   Zulauf_RA_V.Tmr_VZ_Anlauf_Q := TRUE;
   Zulauf_RA_V.SS := FALSE;
   Zulauf_RA_V.SSnq := FALSE;
   Zulauf_RA_V.SSfq := TRUE;
   Zulauf_RA_V.nBB := FALSE;
   Zulauf_RA_V.VW_Hand_St1 := FALSE;
   Zulauf_RA_V.VW_Hand_St2 := FALSE;
   Zulauf_RA_V.VW_Hand_Stop := FALSE;
   Zulauf_RA_V.VW_Auto_St1 := FALSE;
   Zulauf_RA_V.VW_Auto_St2 := FALSE;
   Zulauf_RA_V.Anst_Req_St1 := FALSE;
   Zulauf_RA_V.Anst_Req_St2 := FALSE;
   Zulauf_RA_V.FM_Betrieb_Ein := TRUE;
   Zulauf_RA_V.FM_Betrieb_Aus := FALSE;
   Zulauf_RA_V.NLZ_MAZ_St1 := FALSE;
   Zulauf_RA_V.NLZ_MAZ_St2 := FALSE;
   Zulauf_RA_V.NLZ_Rev_SS_St1 := FALSE;
   Zulauf_RA_V.NLZ_Rev_SS_St2 := FALSE;
   Zulauf_RA_V.Th_St := FALSE;
   Zulauf_RA_V.DMA_St := FALSE;
   Zulauf_RA_V.DMZ_St := FALSE;
   Zulauf_RA_V.FU_St := FALSE;
   Zulauf_RA_V.TL_St := FALSE;
   Zulauf_RA_V.UDr_St := FALSE;
   Zulauf_RA_V.UeDr_St := FALSE;
   Zulauf_RA_V.UT_St := FALSE;
   Zulauf_RA_V.Le_St := FALSE;
   Zulauf_RA_V.UeLM_St := FALSE;
   Zulauf_RA_V.UeLE_St := FALSE;
   Zulauf_RA_V.Kom_DP_St := FALSE;
   Zulauf_RA_V.Kom_int_St := FALSE;
   Zulauf_RA_V.int_St := FALSE;
   Zulauf_RA_V.LZ_St := FALSE;
   Zulauf_RA_V.BefLZ_St := FALSE;
   Zulauf_RA_V.FM_GlobalQuit := FALSE;
   Zulauf_RA_V.Quit_RST := FALSE;
   Zulauf_RA_V.Tmr_VZ_Anlauf := 3;
   Zulauf_RA_V.Tmr_VZ_ESZ := 0;
   Zulauf_RA_V.Tmr_Th_St := 0;
   Zulauf_RA_V.Tmr_DMA_St := 0;
   Zulauf_RA_V.Tmr_DMZ_St := 0;
   Zulauf_RA_V.Tmr_FU_St := 0;
   Zulauf_RA_V.Tmr_TL_St := 0;
   Zulauf_RA_V.Tmr_UDr_St := 0;
   Zulauf_RA_V.Tmr_UeDr_St := 0;
   Zulauf_RA_V.Tmr_UT_St := 0;
   Zulauf_RA_V.Tmr_Le_St := 0;
   Zulauf_RA_V.Tmr_UeLM_St := 0;
   Zulauf_RA_V.Tmr_UeLE_St := 0;
   Zulauf_RA_V.Tmr_Kom_DP_St := 0;
   Zulauf_RA_V.Tmr_Kom_int_St := 0;
   Zulauf_RA_V.Tmr_int_St := 0;
   Zulauf_RA_V.Tmr_LZ_St := 0;
   Zulauf_RA_V.Tmr_BefLZ_St := 0;
   Zulauf_RA_V.Tmr_ASZ_St1 := 0;
   Zulauf_RA_V.Tmr_ASZ_St2 := 0;
   Zulauf_RA_V.Tmr_Rev_St1 := 0;
   Zulauf_RA_V.Tmr_Rev_St2 := 0;
   Zulauf_RA_V.BZ_ges_s := 3248;
   Zulauf_RA_V.Tmr_Quit_RST := 0;
   Zulauf_RA_V.BEF_NHV.Bef.Bed_Res := FALSE;
   Zulauf_RA_V.BEF_NHV.Bef.Bed_UV := FALSE;
   Zulauf_RA_V.BEF_NHV.Bef.Bed_NHV := FALSE;
   Zulauf_RA_V.BEF_NHV.Bef.Bed_PLS := FALSE;
   Zulauf_RA_V.BEF_NHV.Bef.BA_Hand := FALSE;
   Zulauf_RA_V.BEF_NHV.Bef.BA_Auto := FALSE;
   Zulauf_RA_V.BEF_NHV.Bef.BF_Ein1 := FALSE;
   Zulauf_RA_V.BEF_NHV.Bef.BF_Ein2 := FALSE;
   Zulauf_RA_V.BEF_NHV.Bef.BF_Aus := FALSE;
   Zulauf_RA_V.BEF_NHV.Bef.BZ_Res := FALSE;
   Zulauf_RA_V.BEF_NHV.Bef.Res_10 := FALSE;
   Zulauf_RA_V.BEF_NHV.Bef.Res_11 := FALSE;
   Zulauf_RA_V.BEF_NHV.Bef.Res_12 := FALSE;
   Zulauf_RA_V.BEF_NHV.Bef.Res_13 := FALSE;
   Zulauf_RA_V.BEF_NHV.Bef.Res_14 := FALSE;
   Zulauf_RA_V.BEF_NHV.Bef.Res_15 := FALSE;
   Zulauf_RA_V.BEF_NHV.Bef.Res_16 := FALSE;
   Zulauf_RA_V.BEF_NHV.Bef.Res_17 := FALSE;
   Zulauf_RA_V.BEF_NHV.Bef.Res_18 := FALSE;
   Zulauf_RA_V.BEF_NHV.Bef.Res_19 := FALSE;
   Zulauf_RA_V.BEF_NHV.Bef.Res_20 := FALSE;
   Zulauf_RA_V.BEF_NHV.Bef.Res_21 := FALSE;
   Zulauf_RA_V.BEF_NHV.Bef.Res_22 := FALSE;
   Zulauf_RA_V.BEF_NHV.Bef.Res_23 := FALSE;
   Zulauf_RA_V.BEF_NHV.Bef.Res_24 := FALSE;
   Zulauf_RA_V.BEF_NHV.Bef.Res_25 := FALSE;
   Zulauf_RA_V.BEF_NHV.Bef.Res_26 := FALSE;
   Zulauf_RA_V.BEF_NHV.Bef.Res_27 := FALSE;
   Zulauf_RA_V.BEF_NHV.Bef.Res_28 := FALSE;
   Zulauf_RA_V.BEF_NHV.Bef.Res_29 := FALSE;
   Zulauf_RA_V.BEF_NHV.Bef.BF_Set_SW_chg := FALSE;
   Zulauf_RA_V.BEF_NHV.Bef.BF_Quit := FALSE;
   Zulauf_RA_V.BEF_NHV.SW_Hand := 0.0;
   Zulauf_RA_RP.Typ := 0;
   Zulauf_RA_RP.Idx := 31;
   Zulauf_RA_RP.BA_VW_Hand := FALSE;
   Zulauf_RA_RP.Tmr_VZ_Anlauf_Q := FALSE;
   Zulauf_RA_RP.SS := FALSE;
   Zulauf_RA_RP.SSnq := FALSE;
   Zulauf_RA_RP.SSfq := TRUE;
   Zulauf_RA_RP.nBB := FALSE;
   Zulauf_RA_RP.VW_Hand_St1 := FALSE;
   Zulauf_RA_RP.VW_Hand_St2 := FALSE;
   Zulauf_RA_RP.VW_Hand_Stop := FALSE;
   Zulauf_RA_RP.VW_Auto_St1 := FALSE;
   Zulauf_RA_RP.VW_Auto_St2 := FALSE;
   Zulauf_RA_RP.Anst_Req_St1 := FALSE;
   Zulauf_RA_RP.Anst_Req_St2 := FALSE;
   Zulauf_RA_RP.FM_Betrieb_Ein := FALSE;
   Zulauf_RA_RP.FM_Betrieb_Aus := TRUE;
   Zulauf_RA_RP.NLZ_MAZ_St1 := FALSE;
   Zulauf_RA_RP.NLZ_MAZ_St2 := FALSE;
   Zulauf_RA_RP.NLZ_Rev_SS_St1 := FALSE;
   Zulauf_RA_RP.NLZ_Rev_SS_St2 := FALSE;
   Zulauf_RA_RP.Th_St := FALSE;
   Zulauf_RA_RP.DMA_St := FALSE;
   Zulauf_RA_RP.DMZ_St := FALSE;
   Zulauf_RA_RP.FU_St := FALSE;
   Zulauf_RA_RP.TL_St := FALSE;
   Zulauf_RA_RP.UDr_St := FALSE;
   Zulauf_RA_RP.UeDr_St := FALSE;
   Zulauf_RA_RP.UT_St := FALSE;
   Zulauf_RA_RP.Le_St := FALSE;
   Zulauf_RA_RP.UeLM_St := FALSE;
   Zulauf_RA_RP.UeLE_St := FALSE;
   Zulauf_RA_RP.Kom_DP_St := FALSE;
   Zulauf_RA_RP.Kom_int_St := FALSE;
   Zulauf_RA_RP.int_St := FALSE;
   Zulauf_RA_RP.LZ_St := FALSE;
   Zulauf_RA_RP.BefLZ_St := FALSE;
   Zulauf_RA_RP.FM_GlobalQuit := FALSE;
   Zulauf_RA_RP.Quit_RST := FALSE;
   Zulauf_RA_RP.Tmr_VZ_Anlauf := 0;
   Zulauf_RA_RP.Tmr_VZ_ESZ := 0;
   Zulauf_RA_RP.Tmr_Th_St := 0;
   Zulauf_RA_RP.Tmr_DMA_St := 0;
   Zulauf_RA_RP.Tmr_DMZ_St := 0;
   Zulauf_RA_RP.Tmr_FU_St := 0;
   Zulauf_RA_RP.Tmr_TL_St := 0;
   Zulauf_RA_RP.Tmr_UDr_St := 0;
   Zulauf_RA_RP.Tmr_UeDr_St := 0;
   Zulauf_RA_RP.Tmr_UT_St := 0;
   Zulauf_RA_RP.Tmr_Le_St := 0;
   Zulauf_RA_RP.Tmr_UeLM_St := 0;
   Zulauf_RA_RP.Tmr_UeLE_St := 0;
   Zulauf_RA_RP.Tmr_Kom_DP_St := 0;
   Zulauf_RA_RP.Tmr_Kom_int_St := 0;
   Zulauf_RA_RP.Tmr_int_St := 0;
   Zulauf_RA_RP.Tmr_LZ_St := 0;
   Zulauf_RA_RP.Tmr_BefLZ_St := 0;
   Zulauf_RA_RP.Tmr_ASZ_St1 := 0;
   Zulauf_RA_RP.Tmr_ASZ_St2 := 0;
   Zulauf_RA_RP.Tmr_Rev_St1 := 0;
   Zulauf_RA_RP.Tmr_Rev_St2 := 0;
   Zulauf_RA_RP.BZ_ges_s := 455;
   Zulauf_RA_RP.Tmr_Quit_RST := 0;
   Zulauf_RA_RP.BEF_NHV.Bef.Bed_Res := FALSE;
   Zulauf_RA_RP.BEF_NHV.Bef.Bed_UV := FALSE;
   Zulauf_RA_RP.BEF_NHV.Bef.Bed_NHV := FALSE;
   Zulauf_RA_RP.BEF_NHV.Bef.Bed_PLS := FALSE;
   Zulauf_RA_RP.BEF_NHV.Bef.BA_Hand := FALSE;
   Zulauf_RA_RP.BEF_NHV.Bef.BA_Auto := FALSE;
   Zulauf_RA_RP.BEF_NHV.Bef.BF_Ein1 := FALSE;
   Zulauf_RA_RP.BEF_NHV.Bef.BF_Ein2 := FALSE;
   Zulauf_RA_RP.BEF_NHV.Bef.BF_Aus := FALSE;
   Zulauf_RA_RP.BEF_NHV.Bef.BZ_Res := FALSE;
   Zulauf_RA_RP.BEF_NHV.Bef.Res_10 := FALSE;
   Zulauf_RA_RP.BEF_NHV.Bef.Res_11 := FALSE;
   Zulauf_RA_RP.BEF_NHV.Bef.Res_12 := FALSE;
   Zulauf_RA_RP.BEF_NHV.Bef.Res_13 := FALSE;
   Zulauf_RA_RP.BEF_NHV.Bef.Res_14 := FALSE;
   Zulauf_RA_RP.BEF_NHV.Bef.Res_15 := FALSE;
   Zulauf_RA_RP.BEF_NHV.Bef.Res_16 := FALSE;
   Zulauf_RA_RP.BEF_NHV.Bef.Res_17 := FALSE;
   Zulauf_RA_RP.BEF_NHV.Bef.Res_18 := FALSE;
   Zulauf_RA_RP.BEF_NHV.Bef.Res_19 := FALSE;
   Zulauf_RA_RP.BEF_NHV.Bef.Res_20 := FALSE;
   Zulauf_RA_RP.BEF_NHV.Bef.Res_21 := FALSE;
   Zulauf_RA_RP.BEF_NHV.Bef.Res_22 := FALSE;
   Zulauf_RA_RP.BEF_NHV.Bef.Res_23 := FALSE;
   Zulauf_RA_RP.BEF_NHV.Bef.Res_24 := FALSE;
   Zulauf_RA_RP.BEF_NHV.Bef.Res_25 := FALSE;
   Zulauf_RA_RP.BEF_NHV.Bef.Res_26 := FALSE;
   Zulauf_RA_RP.BEF_NHV.Bef.Res_27 := FALSE;
   Zulauf_RA_RP.BEF_NHV.Bef.Res_28 := FALSE;
   Zulauf_RA_RP.BEF_NHV.Bef.Res_29 := FALSE;
   Zulauf_RA_RP.BEF_NHV.Bef.BF_Set_SW_chg := FALSE;
   Zulauf_RA_RP.BEF_NHV.Bef.BF_Quit := FALSE;
   Zulauf_RA_RP.BEF_NHV.SW_Hand := 0.0;
   Zulauf_RA_FP.Typ := 0;
   Zulauf_RA_FP.Idx := 32;
   Zulauf_RA_FP.BA_VW_Hand := FALSE;
   Zulauf_RA_FP.Tmr_VZ_Anlauf_Q := FALSE;
   Zulauf_RA_FP.SS := FALSE;
   Zulauf_RA_FP.SSnq := FALSE;
   Zulauf_RA_FP.SSfq := TRUE;
   Zulauf_RA_FP.nBB := FALSE;
   Zulauf_RA_FP.VW_Hand_St1 := FALSE;
   Zulauf_RA_FP.VW_Hand_St2 := FALSE;
   Zulauf_RA_FP.VW_Hand_Stop := FALSE;
   Zulauf_RA_FP.VW_Auto_St1 := FALSE;
   Zulauf_RA_FP.VW_Auto_St2 := FALSE;
   Zulauf_RA_FP.Anst_Req_St1 := FALSE;
   Zulauf_RA_FP.Anst_Req_St2 := FALSE;
   Zulauf_RA_FP.FM_Betrieb_Ein := FALSE;
   Zulauf_RA_FP.FM_Betrieb_Aus := TRUE;
   Zulauf_RA_FP.NLZ_MAZ_St1 := FALSE;
   Zulauf_RA_FP.NLZ_MAZ_St2 := FALSE;
   Zulauf_RA_FP.NLZ_Rev_SS_St1 := FALSE;
   Zulauf_RA_FP.NLZ_Rev_SS_St2 := FALSE;
   Zulauf_RA_FP.Th_St := FALSE;
   Zulauf_RA_FP.DMA_St := FALSE;
   Zulauf_RA_FP.DMZ_St := FALSE;
   Zulauf_RA_FP.FU_St := FALSE;
   Zulauf_RA_FP.TL_St := FALSE;
   Zulauf_RA_FP.UDr_St := FALSE;
   Zulauf_RA_FP.UeDr_St := FALSE;
   Zulauf_RA_FP.UT_St := FALSE;
   Zulauf_RA_FP.Le_St := FALSE;
   Zulauf_RA_FP.UeLM_St := FALSE;
   Zulauf_RA_FP.UeLE_St := FALSE;
   Zulauf_RA_FP.Kom_DP_St := FALSE;
   Zulauf_RA_FP.Kom_int_St := FALSE;
   Zulauf_RA_FP.int_St := FALSE;
   Zulauf_RA_FP.LZ_St := FALSE;
   Zulauf_RA_FP.BefLZ_St := FALSE;
   Zulauf_RA_FP.FM_GlobalQuit := FALSE;
   Zulauf_RA_FP.Quit_RST := FALSE;
   Zulauf_RA_FP.Tmr_VZ_Anlauf := 0;
   Zulauf_RA_FP.Tmr_VZ_ESZ := 0;
   Zulauf_RA_FP.Tmr_Th_St := 0;
   Zulauf_RA_FP.Tmr_DMA_St := 0;
   Zulauf_RA_FP.Tmr_DMZ_St := 0;
   Zulauf_RA_FP.Tmr_FU_St := 0;
   Zulauf_RA_FP.Tmr_TL_St := 0;
   Zulauf_RA_FP.Tmr_UDr_St := 0;
   Zulauf_RA_FP.Tmr_UeDr_St := 0;
   Zulauf_RA_FP.Tmr_UT_St := 0;
   Zulauf_RA_FP.Tmr_Le_St := 0;
   Zulauf_RA_FP.Tmr_UeLM_St := 0;
   Zulauf_RA_FP.Tmr_UeLE_St := 0;
   Zulauf_RA_FP.Tmr_Kom_DP_St := 0;
   Zulauf_RA_FP.Tmr_Kom_int_St := 0;
   Zulauf_RA_FP.Tmr_int_St := 0;
   Zulauf_RA_FP.Tmr_LZ_St := 0;
   Zulauf_RA_FP.Tmr_BefLZ_St := 0;
   Zulauf_RA_FP.Tmr_ASZ_St1 := 0;
   Zulauf_RA_FP.Tmr_ASZ_St2 := 0;
   Zulauf_RA_FP.Tmr_Rev_St1 := 0;
   Zulauf_RA_FP.Tmr_Rev_St2 := 0;
   Zulauf_RA_FP.BZ_ges_s := 701;
   Zulauf_RA_FP.Tmr_Quit_RST := 0;
   Zulauf_RA_FP.BEF_NHV.Bef.Bed_Res := FALSE;
   Zulauf_RA_FP.BEF_NHV.Bef.Bed_UV := FALSE;
   Zulauf_RA_FP.BEF_NHV.Bef.Bed_NHV := FALSE;
   Zulauf_RA_FP.BEF_NHV.Bef.Bed_PLS := FALSE;
   Zulauf_RA_FP.BEF_NHV.Bef.BA_Hand := FALSE;
   Zulauf_RA_FP.BEF_NHV.Bef.BA_Auto := FALSE;
   Zulauf_RA_FP.BEF_NHV.Bef.BF_Ein1 := FALSE;
   Zulauf_RA_FP.BEF_NHV.Bef.BF_Ein2 := FALSE;
   Zulauf_RA_FP.BEF_NHV.Bef.BF_Aus := FALSE;
   Zulauf_RA_FP.BEF_NHV.Bef.BZ_Res := FALSE;
   Zulauf_RA_FP.BEF_NHV.Bef.Res_10 := FALSE;
   Zulauf_RA_FP.BEF_NHV.Bef.Res_11 := FALSE;
   Zulauf_RA_FP.BEF_NHV.Bef.Res_12 := FALSE;
   Zulauf_RA_FP.BEF_NHV.Bef.Res_13 := FALSE;
   Zulauf_RA_FP.BEF_NHV.Bef.Res_14 := FALSE;
   Zulauf_RA_FP.BEF_NHV.Bef.Res_15 := FALSE;
   Zulauf_RA_FP.BEF_NHV.Bef.Res_16 := FALSE;
   Zulauf_RA_FP.BEF_NHV.Bef.Res_17 := FALSE;
   Zulauf_RA_FP.BEF_NHV.Bef.Res_18 := FALSE;
   Zulauf_RA_FP.BEF_NHV.Bef.Res_19 := FALSE;
   Zulauf_RA_FP.BEF_NHV.Bef.Res_20 := FALSE;
   Zulauf_RA_FP.BEF_NHV.Bef.Res_21 := FALSE;
   Zulauf_RA_FP.BEF_NHV.Bef.Res_22 := FALSE;
   Zulauf_RA_FP.BEF_NHV.Bef.Res_23 := FALSE;
   Zulauf_RA_FP.BEF_NHV.Bef.Res_24 := FALSE;
   Zulauf_RA_FP.BEF_NHV.Bef.Res_25 := FALSE;
   Zulauf_RA_FP.BEF_NHV.Bef.Res_26 := FALSE;
   Zulauf_RA_FP.BEF_NHV.Bef.Res_27 := FALSE;
   Zulauf_RA_FP.BEF_NHV.Bef.Res_28 := FALSE;
   Zulauf_RA_FP.BEF_NHV.Bef.Res_29 := FALSE;
   Zulauf_RA_FP.BEF_NHV.Bef.BF_Set_SW_chg := FALSE;
   Zulauf_RA_FP.BEF_NHV.Bef.BF_Quit := FALSE;
   Zulauf_RA_FP.BEF_NHV.SW_Hand := 0.0;
   Schlamm_BP.Typ := 0;
   Schlamm_BP.Idx := 33;
   Schlamm_BP.BA_VW_Hand := FALSE;
   Schlamm_BP.Tmr_VZ_Anlauf_Q := FALSE;
   Schlamm_BP.SS := FALSE;
   Schlamm_BP.SSnq := FALSE;
   Schlamm_BP.SSfq := TRUE;
   Schlamm_BP.nBB := FALSE;
   Schlamm_BP.VW_Hand_St1 := FALSE;
   Schlamm_BP.VW_Hand_St2 := FALSE;
   Schlamm_BP.VW_Hand_Stop := FALSE;
   Schlamm_BP.VW_Auto_St1 := FALSE;
   Schlamm_BP.VW_Auto_St2 := FALSE;
   Schlamm_BP.Anst_Req_St1 := FALSE;
   Schlamm_BP.Anst_Req_St2 := FALSE;
   Schlamm_BP.FM_Betrieb_Ein := FALSE;
   Schlamm_BP.FM_Betrieb_Aus := TRUE;
   Schlamm_BP.NLZ_MAZ_St1 := FALSE;
   Schlamm_BP.NLZ_MAZ_St2 := FALSE;
   Schlamm_BP.NLZ_Rev_SS_St1 := FALSE;
   Schlamm_BP.NLZ_Rev_SS_St2 := FALSE;
   Schlamm_BP.Th_St := FALSE;
   Schlamm_BP.DMA_St := FALSE;
   Schlamm_BP.DMZ_St := FALSE;
   Schlamm_BP.FU_St := FALSE;
   Schlamm_BP.TL_St := FALSE;
   Schlamm_BP.UDr_St := FALSE;
   Schlamm_BP.UeDr_St := FALSE;
   Schlamm_BP.UT_St := FALSE;
   Schlamm_BP.Le_St := FALSE;
   Schlamm_BP.UeLM_St := FALSE;
   Schlamm_BP.UeLE_St := FALSE;
   Schlamm_BP.Kom_DP_St := FALSE;
   Schlamm_BP.Kom_int_St := FALSE;
   Schlamm_BP.int_St := FALSE;
   Schlamm_BP.LZ_St := FALSE;
   Schlamm_BP.BefLZ_St := FALSE;
   Schlamm_BP.FM_GlobalQuit := FALSE;
   Schlamm_BP.Quit_RST := FALSE;
   Schlamm_BP.Tmr_VZ_Anlauf := 0;
   Schlamm_BP.Tmr_VZ_ESZ := 0;
   Schlamm_BP.Tmr_Th_St := 0;
   Schlamm_BP.Tmr_DMA_St := 0;
   Schlamm_BP.Tmr_DMZ_St := 0;
   Schlamm_BP.Tmr_FU_St := 0;
   Schlamm_BP.Tmr_TL_St := 0;
   Schlamm_BP.Tmr_UDr_St := 0;
   Schlamm_BP.Tmr_UeDr_St := 0;
   Schlamm_BP.Tmr_UT_St := 0;
   Schlamm_BP.Tmr_Le_St := 0;
   Schlamm_BP.Tmr_UeLM_St := 0;
   Schlamm_BP.Tmr_UeLE_St := 0;
   Schlamm_BP.Tmr_Kom_DP_St := 0;
   Schlamm_BP.Tmr_Kom_int_St := 0;
   Schlamm_BP.Tmr_int_St := 0;
   Schlamm_BP.Tmr_LZ_St := 0;
   Schlamm_BP.Tmr_BefLZ_St := 0;
   Schlamm_BP.Tmr_ASZ_St1 := 0;
   Schlamm_BP.Tmr_ASZ_St2 := 0;
   Schlamm_BP.Tmr_Rev_St1 := 0;
   Schlamm_BP.Tmr_Rev_St2 := 0;
   Schlamm_BP.BZ_ges_s := 708;
   Schlamm_BP.Tmr_Quit_RST := 0;
   Schlamm_BP.BEF_NHV.Bef.Bed_Res := FALSE;
   Schlamm_BP.BEF_NHV.Bef.Bed_UV := FALSE;
   Schlamm_BP.BEF_NHV.Bef.Bed_NHV := FALSE;
   Schlamm_BP.BEF_NHV.Bef.Bed_PLS := FALSE;
   Schlamm_BP.BEF_NHV.Bef.BA_Hand := FALSE;
   Schlamm_BP.BEF_NHV.Bef.BA_Auto := FALSE;
   Schlamm_BP.BEF_NHV.Bef.BF_Ein1 := FALSE;
   Schlamm_BP.BEF_NHV.Bef.BF_Ein2 := FALSE;
   Schlamm_BP.BEF_NHV.Bef.BF_Aus := FALSE;
   Schlamm_BP.BEF_NHV.Bef.BZ_Res := FALSE;
   Schlamm_BP.BEF_NHV.Bef.Res_10 := FALSE;
   Schlamm_BP.BEF_NHV.Bef.Res_11 := FALSE;
   Schlamm_BP.BEF_NHV.Bef.Res_12 := FALSE;
   Schlamm_BP.BEF_NHV.Bef.Res_13 := FALSE;
   Schlamm_BP.BEF_NHV.Bef.Res_14 := FALSE;
   Schlamm_BP.BEF_NHV.Bef.Res_15 := FALSE;
   Schlamm_BP.BEF_NHV.Bef.Res_16 := FALSE;
   Schlamm_BP.BEF_NHV.Bef.Res_17 := FALSE;
   Schlamm_BP.BEF_NHV.Bef.Res_18 := FALSE;
   Schlamm_BP.BEF_NHV.Bef.Res_19 := FALSE;
   Schlamm_BP.BEF_NHV.Bef.Res_20 := FALSE;
   Schlamm_BP.BEF_NHV.Bef.Res_21 := FALSE;
   Schlamm_BP.BEF_NHV.Bef.Res_22 := FALSE;
   Schlamm_BP.BEF_NHV.Bef.Res_23 := FALSE;
   Schlamm_BP.BEF_NHV.Bef.Res_24 := FALSE;
   Schlamm_BP.BEF_NHV.Bef.Res_25 := FALSE;
   Schlamm_BP.BEF_NHV.Bef.Res_26 := FALSE;
   Schlamm_BP.BEF_NHV.Bef.Res_27 := FALSE;
   Schlamm_BP.BEF_NHV.Bef.Res_28 := FALSE;
   Schlamm_BP.BEF_NHV.Bef.Res_29 := FALSE;
   Schlamm_BP.BEF_NHV.Bef.BF_Set_SW_chg := FALSE;
   Schlamm_BP.BEF_NHV.Bef.BF_Quit := FALSE;
   Schlamm_BP.BEF_NHV.SW_Hand := 0.0;
   Truebwasser_P1.Typ := 0;
   Truebwasser_P1.Idx := 34;
   Truebwasser_P1.BA_VW_Hand := FALSE;
   Truebwasser_P1.Tmr_VZ_Anlauf_Q := FALSE;
   Truebwasser_P1.SS := FALSE;
   Truebwasser_P1.SSnq := FALSE;
   Truebwasser_P1.SSfq := TRUE;
   Truebwasser_P1.nBB := FALSE;
   Truebwasser_P1.VW_Hand_St1 := FALSE;
   Truebwasser_P1.VW_Hand_St2 := FALSE;
   Truebwasser_P1.VW_Hand_Stop := FALSE;
   Truebwasser_P1.VW_Auto_St1 := FALSE;
   Truebwasser_P1.VW_Auto_St2 := FALSE;
   Truebwasser_P1.Anst_Req_St1 := FALSE;
   Truebwasser_P1.Anst_Req_St2 := FALSE;
   Truebwasser_P1.FM_Betrieb_Ein := FALSE;
   Truebwasser_P1.FM_Betrieb_Aus := TRUE;
   Truebwasser_P1.NLZ_MAZ_St1 := FALSE;
   Truebwasser_P1.NLZ_MAZ_St2 := FALSE;
   Truebwasser_P1.NLZ_Rev_SS_St1 := FALSE;
   Truebwasser_P1.NLZ_Rev_SS_St2 := FALSE;
   Truebwasser_P1.Th_St := FALSE;
   Truebwasser_P1.DMA_St := FALSE;
   Truebwasser_P1.DMZ_St := FALSE;
   Truebwasser_P1.FU_St := FALSE;
   Truebwasser_P1.TL_St := FALSE;
   Truebwasser_P1.UDr_St := FALSE;
   Truebwasser_P1.UeDr_St := FALSE;
   Truebwasser_P1.UT_St := FALSE;
   Truebwasser_P1.Le_St := FALSE;
   Truebwasser_P1.UeLM_St := FALSE;
   Truebwasser_P1.UeLE_St := FALSE;
   Truebwasser_P1.Kom_DP_St := FALSE;
   Truebwasser_P1.Kom_int_St := FALSE;
   Truebwasser_P1.int_St := FALSE;
   Truebwasser_P1.LZ_St := FALSE;
   Truebwasser_P1.BefLZ_St := FALSE;
   Truebwasser_P1.FM_GlobalQuit := FALSE;
   Truebwasser_P1.Quit_RST := FALSE;
   Truebwasser_P1.Tmr_VZ_Anlauf := 0;
   Truebwasser_P1.Tmr_VZ_ESZ := 0;
   Truebwasser_P1.Tmr_Th_St := 0;
   Truebwasser_P1.Tmr_DMA_St := 0;
   Truebwasser_P1.Tmr_DMZ_St := 0;
   Truebwasser_P1.Tmr_FU_St := 0;
   Truebwasser_P1.Tmr_TL_St := 0;
   Truebwasser_P1.Tmr_UDr_St := 0;
   Truebwasser_P1.Tmr_UeDr_St := 0;
   Truebwasser_P1.Tmr_UT_St := 0;
   Truebwasser_P1.Tmr_Le_St := 0;
   Truebwasser_P1.Tmr_UeLM_St := 0;
   Truebwasser_P1.Tmr_UeLE_St := 0;
   Truebwasser_P1.Tmr_Kom_DP_St := 0;
   Truebwasser_P1.Tmr_Kom_int_St := 0;
   Truebwasser_P1.Tmr_int_St := 0;
   Truebwasser_P1.Tmr_LZ_St := 0;
   Truebwasser_P1.Tmr_BefLZ_St := 0;
   Truebwasser_P1.Tmr_ASZ_St1 := 0;
   Truebwasser_P1.Tmr_ASZ_St2 := 0;
   Truebwasser_P1.Tmr_Rev_St1 := 0;
   Truebwasser_P1.Tmr_Rev_St2 := 0;
   Truebwasser_P1.BZ_ges_s := 842;
   Truebwasser_P1.Tmr_Quit_RST := 0;
   Truebwasser_P1.BEF_NHV.Bef.Bed_Res := FALSE;
   Truebwasser_P1.BEF_NHV.Bef.Bed_UV := FALSE;
   Truebwasser_P1.BEF_NHV.Bef.Bed_NHV := FALSE;
   Truebwasser_P1.BEF_NHV.Bef.Bed_PLS := FALSE;
   Truebwasser_P1.BEF_NHV.Bef.BA_Hand := FALSE;
   Truebwasser_P1.BEF_NHV.Bef.BA_Auto := FALSE;
   Truebwasser_P1.BEF_NHV.Bef.BF_Ein1 := FALSE;
   Truebwasser_P1.BEF_NHV.Bef.BF_Ein2 := FALSE;
   Truebwasser_P1.BEF_NHV.Bef.BF_Aus := FALSE;
   Truebwasser_P1.BEF_NHV.Bef.BZ_Res := FALSE;
   Truebwasser_P1.BEF_NHV.Bef.Res_10 := FALSE;
   Truebwasser_P1.BEF_NHV.Bef.Res_11 := FALSE;
   Truebwasser_P1.BEF_NHV.Bef.Res_12 := FALSE;
   Truebwasser_P1.BEF_NHV.Bef.Res_13 := FALSE;
   Truebwasser_P1.BEF_NHV.Bef.Res_14 := FALSE;
   Truebwasser_P1.BEF_NHV.Bef.Res_15 := FALSE;
   Truebwasser_P1.BEF_NHV.Bef.Res_16 := FALSE;
   Truebwasser_P1.BEF_NHV.Bef.Res_17 := FALSE;
   Truebwasser_P1.BEF_NHV.Bef.Res_18 := FALSE;
   Truebwasser_P1.BEF_NHV.Bef.Res_19 := FALSE;
   Truebwasser_P1.BEF_NHV.Bef.Res_20 := FALSE;
   Truebwasser_P1.BEF_NHV.Bef.Res_21 := FALSE;
   Truebwasser_P1.BEF_NHV.Bef.Res_22 := FALSE;
   Truebwasser_P1.BEF_NHV.Bef.Res_23 := FALSE;
   Truebwasser_P1.BEF_NHV.Bef.Res_24 := FALSE;
   Truebwasser_P1.BEF_NHV.Bef.Res_25 := FALSE;
   Truebwasser_P1.BEF_NHV.Bef.Res_26 := FALSE;
   Truebwasser_P1.BEF_NHV.Bef.Res_27 := FALSE;
   Truebwasser_P1.BEF_NHV.Bef.Res_28 := FALSE;
   Truebwasser_P1.BEF_NHV.Bef.Res_29 := FALSE;
   Truebwasser_P1.BEF_NHV.Bef.BF_Set_SW_chg := FALSE;
   Truebwasser_P1.BEF_NHV.Bef.BF_Quit := FALSE;
   Truebwasser_P1.BEF_NHV.SW_Hand := 0.0;
   Truebwasser_P2.Typ := 0;
   Truebwasser_P2.Idx := 35;
   Truebwasser_P2.BA_VW_Hand := FALSE;
   Truebwasser_P2.Tmr_VZ_Anlauf_Q := FALSE;
   Truebwasser_P2.SS := FALSE;
   Truebwasser_P2.SSnq := FALSE;
   Truebwasser_P2.SSfq := TRUE;
   Truebwasser_P2.nBB := FALSE;
   Truebwasser_P2.VW_Hand_St1 := FALSE;
   Truebwasser_P2.VW_Hand_St2 := FALSE;
   Truebwasser_P2.VW_Hand_Stop := FALSE;
   Truebwasser_P2.VW_Auto_St1 := FALSE;
   Truebwasser_P2.VW_Auto_St2 := FALSE;
   Truebwasser_P2.Anst_Req_St1 := FALSE;
   Truebwasser_P2.Anst_Req_St2 := FALSE;
   Truebwasser_P2.FM_Betrieb_Ein := FALSE;
   Truebwasser_P2.FM_Betrieb_Aus := TRUE;
   Truebwasser_P2.NLZ_MAZ_St1 := FALSE;
   Truebwasser_P2.NLZ_MAZ_St2 := FALSE;
   Truebwasser_P2.NLZ_Rev_SS_St1 := FALSE;
   Truebwasser_P2.NLZ_Rev_SS_St2 := FALSE;
   Truebwasser_P2.Th_St := FALSE;
   Truebwasser_P2.DMA_St := FALSE;
   Truebwasser_P2.DMZ_St := FALSE;
   Truebwasser_P2.FU_St := FALSE;
   Truebwasser_P2.TL_St := FALSE;
   Truebwasser_P2.UDr_St := FALSE;
   Truebwasser_P2.UeDr_St := FALSE;
   Truebwasser_P2.UT_St := FALSE;
   Truebwasser_P2.Le_St := FALSE;
   Truebwasser_P2.UeLM_St := FALSE;
   Truebwasser_P2.UeLE_St := FALSE;
   Truebwasser_P2.Kom_DP_St := FALSE;
   Truebwasser_P2.Kom_int_St := FALSE;
   Truebwasser_P2.int_St := FALSE;
   Truebwasser_P2.LZ_St := FALSE;
   Truebwasser_P2.BefLZ_St := FALSE;
   Truebwasser_P2.FM_GlobalQuit := FALSE;
   Truebwasser_P2.Quit_RST := FALSE;
   Truebwasser_P2.Tmr_VZ_Anlauf := 0;
   Truebwasser_P2.Tmr_VZ_ESZ := 0;
   Truebwasser_P2.Tmr_Th_St := 0;
   Truebwasser_P2.Tmr_DMA_St := 0;
   Truebwasser_P2.Tmr_DMZ_St := 0;
   Truebwasser_P2.Tmr_FU_St := 0;
   Truebwasser_P2.Tmr_TL_St := 0;
   Truebwasser_P2.Tmr_UDr_St := 0;
   Truebwasser_P2.Tmr_UeDr_St := 0;
   Truebwasser_P2.Tmr_UT_St := 0;
   Truebwasser_P2.Tmr_Le_St := 0;
   Truebwasser_P2.Tmr_UeLM_St := 0;
   Truebwasser_P2.Tmr_UeLE_St := 0;
   Truebwasser_P2.Tmr_Kom_DP_St := 0;
   Truebwasser_P2.Tmr_Kom_int_St := 0;
   Truebwasser_P2.Tmr_int_St := 0;
   Truebwasser_P2.Tmr_LZ_St := 0;
   Truebwasser_P2.Tmr_BefLZ_St := 0;
   Truebwasser_P2.Tmr_ASZ_St1 := 0;
   Truebwasser_P2.Tmr_ASZ_St2 := 0;
   Truebwasser_P2.Tmr_Rev_St1 := 0;
   Truebwasser_P2.Tmr_Rev_St2 := 0;
   Truebwasser_P2.BZ_ges_s := 1903;
   Truebwasser_P2.Tmr_Quit_RST := 0;
   Truebwasser_P2.BEF_NHV.Bef.Bed_Res := FALSE;
   Truebwasser_P2.BEF_NHV.Bef.Bed_UV := FALSE;
   Truebwasser_P2.BEF_NHV.Bef.Bed_NHV := FALSE;
   Truebwasser_P2.BEF_NHV.Bef.Bed_PLS := FALSE;
   Truebwasser_P2.BEF_NHV.Bef.BA_Hand := FALSE;
   Truebwasser_P2.BEF_NHV.Bef.BA_Auto := FALSE;
   Truebwasser_P2.BEF_NHV.Bef.BF_Ein1 := FALSE;
   Truebwasser_P2.BEF_NHV.Bef.BF_Ein2 := FALSE;
   Truebwasser_P2.BEF_NHV.Bef.BF_Aus := FALSE;
   Truebwasser_P2.BEF_NHV.Bef.BZ_Res := FALSE;
   Truebwasser_P2.BEF_NHV.Bef.Res_10 := FALSE;
   Truebwasser_P2.BEF_NHV.Bef.Res_11 := FALSE;
   Truebwasser_P2.BEF_NHV.Bef.Res_12 := FALSE;
   Truebwasser_P2.BEF_NHV.Bef.Res_13 := FALSE;
   Truebwasser_P2.BEF_NHV.Bef.Res_14 := FALSE;
   Truebwasser_P2.BEF_NHV.Bef.Res_15 := FALSE;
   Truebwasser_P2.BEF_NHV.Bef.Res_16 := FALSE;
   Truebwasser_P2.BEF_NHV.Bef.Res_17 := FALSE;
   Truebwasser_P2.BEF_NHV.Bef.Res_18 := FALSE;
   Truebwasser_P2.BEF_NHV.Bef.Res_19 := FALSE;
   Truebwasser_P2.BEF_NHV.Bef.Res_20 := FALSE;
   Truebwasser_P2.BEF_NHV.Bef.Res_21 := FALSE;
   Truebwasser_P2.BEF_NHV.Bef.Res_22 := FALSE;
   Truebwasser_P2.BEF_NHV.Bef.Res_23 := FALSE;
   Truebwasser_P2.BEF_NHV.Bef.Res_24 := FALSE;
   Truebwasser_P2.BEF_NHV.Bef.Res_25 := FALSE;
   Truebwasser_P2.BEF_NHV.Bef.Res_26 := FALSE;
   Truebwasser_P2.BEF_NHV.Bef.Res_27 := FALSE;
   Truebwasser_P2.BEF_NHV.Bef.Res_28 := FALSE;
   Truebwasser_P2.BEF_NHV.Bef.Res_29 := FALSE;
   Truebwasser_P2.BEF_NHV.Bef.BF_Set_SW_chg := FALSE;
   Truebwasser_P2.BEF_NHV.Bef.BF_Quit := FALSE;
   Truebwasser_P2.BEF_NHV.SW_Hand := 0.0;
   Schlamm_AS.Typ := 5;
   Schlamm_AS.Idx := 36;
   Schlamm_AS.BA_VW_Hand := FALSE;
   Schlamm_AS.Tmr_VZ_Anlauf_Q := FALSE;
   Schlamm_AS.SS := FALSE;
   Schlamm_AS.SSnq := FALSE;
   Schlamm_AS.SSfq := TRUE;
   Schlamm_AS.nBB := FALSE;
   Schlamm_AS.VW_Hand_St1 := FALSE;
   Schlamm_AS.VW_Hand_St2 := FALSE;
   Schlamm_AS.VW_Hand_Stop := FALSE;
   Schlamm_AS.VW_Auto_St1 := FALSE;
   Schlamm_AS.VW_Auto_St2 := FALSE;
   Schlamm_AS.Anst_Req_St1 := FALSE;
   Schlamm_AS.Anst_Req_St2 := FALSE;
   Schlamm_AS.FM_Betrieb_Ein := FALSE;
   Schlamm_AS.FM_Betrieb_Aus := TRUE;
   Schlamm_AS.NLZ_MAZ_St1 := FALSE;
   Schlamm_AS.NLZ_MAZ_St2 := FALSE;
   Schlamm_AS.NLZ_Rev_SS_St1 := FALSE;
   Schlamm_AS.NLZ_Rev_SS_St2 := FALSE;
   Schlamm_AS.Th_St := FALSE;
   Schlamm_AS.DMA_St := FALSE;
   Schlamm_AS.DMZ_St := FALSE;
   Schlamm_AS.FU_St := FALSE;
   Schlamm_AS.TL_St := FALSE;
   Schlamm_AS.UDr_St := FALSE;
   Schlamm_AS.UeDr_St := FALSE;
   Schlamm_AS.UT_St := FALSE;
   Schlamm_AS.Le_St := FALSE;
   Schlamm_AS.UeLM_St := FALSE;
   Schlamm_AS.UeLE_St := FALSE;
   Schlamm_AS.Kom_DP_St := FALSE;
   Schlamm_AS.Kom_int_St := FALSE;
   Schlamm_AS.int_St := FALSE;
   Schlamm_AS.LZ_St := FALSE;
   Schlamm_AS.BefLZ_St := FALSE;
   Schlamm_AS.FM_GlobalQuit := FALSE;
   Schlamm_AS.Quit_RST := FALSE;
   Schlamm_AS.Tmr_VZ_Anlauf := 0;
   Schlamm_AS.Tmr_VZ_ESZ := 0;
   Schlamm_AS.Tmr_Th_St := 0;
   Schlamm_AS.Tmr_DMA_St := 0;
   Schlamm_AS.Tmr_DMZ_St := 0;
   Schlamm_AS.Tmr_FU_St := 0;
   Schlamm_AS.Tmr_TL_St := 0;
   Schlamm_AS.Tmr_UDr_St := 0;
   Schlamm_AS.Tmr_UeDr_St := 0;
   Schlamm_AS.Tmr_UT_St := 0;
   Schlamm_AS.Tmr_Le_St := 0;
   Schlamm_AS.Tmr_UeLM_St := 0;
   Schlamm_AS.Tmr_UeLE_St := 0;
   Schlamm_AS.Tmr_Kom_DP_St := 0;
   Schlamm_AS.Tmr_Kom_int_St := 0;
   Schlamm_AS.Tmr_int_St := 0;
   Schlamm_AS.Tmr_LZ_St := 0;
   Schlamm_AS.Tmr_BefLZ_St := 0;
   Schlamm_AS.Tmr_ASZ_St1 := 0;
   Schlamm_AS.Tmr_ASZ_St2 := 0;
   Schlamm_AS.Tmr_Rev_St1 := 0;
   Schlamm_AS.Tmr_Rev_St2 := 0;
   Schlamm_AS.BZ_ges_s := 139;
   Schlamm_AS.Tmr_Quit_RST := 0;
   Schlamm_AS.BEF_NHV.Bef.Bed_Res := FALSE;
   Schlamm_AS.BEF_NHV.Bef.Bed_UV := FALSE;
   Schlamm_AS.BEF_NHV.Bef.Bed_NHV := FALSE;
   Schlamm_AS.BEF_NHV.Bef.Bed_PLS := FALSE;
   Schlamm_AS.BEF_NHV.Bef.BA_Hand := FALSE;
   Schlamm_AS.BEF_NHV.Bef.BA_Auto := FALSE;
   Schlamm_AS.BEF_NHV.Bef.BF_Ein1 := FALSE;
   Schlamm_AS.BEF_NHV.Bef.BF_Ein2 := FALSE;
   Schlamm_AS.BEF_NHV.Bef.BF_Aus := FALSE;
   Schlamm_AS.BEF_NHV.Bef.BZ_Res := FALSE;
   Schlamm_AS.BEF_NHV.Bef.Res_10 := FALSE;
   Schlamm_AS.BEF_NHV.Bef.Res_11 := FALSE;
   Schlamm_AS.BEF_NHV.Bef.Res_12 := FALSE;
   Schlamm_AS.BEF_NHV.Bef.Res_13 := FALSE;
   Schlamm_AS.BEF_NHV.Bef.Res_14 := FALSE;
   Schlamm_AS.BEF_NHV.Bef.Res_15 := FALSE;
   Schlamm_AS.BEF_NHV.Bef.Res_16 := FALSE;
   Schlamm_AS.BEF_NHV.Bef.Res_17 := FALSE;
   Schlamm_AS.BEF_NHV.Bef.Res_18 := FALSE;
   Schlamm_AS.BEF_NHV.Bef.Res_19 := FALSE;
   Schlamm_AS.BEF_NHV.Bef.Res_20 := FALSE;
   Schlamm_AS.BEF_NHV.Bef.Res_21 := FALSE;
   Schlamm_AS.BEF_NHV.Bef.Res_22 := FALSE;
   Schlamm_AS.BEF_NHV.Bef.Res_23 := FALSE;
   Schlamm_AS.BEF_NHV.Bef.Res_24 := FALSE;
   Schlamm_AS.BEF_NHV.Bef.Res_25 := FALSE;
   Schlamm_AS.BEF_NHV.Bef.Res_26 := FALSE;
   Schlamm_AS.BEF_NHV.Bef.Res_27 := FALSE;
   Schlamm_AS.BEF_NHV.Bef.Res_28 := FALSE;
   Schlamm_AS.BEF_NHV.Bef.Res_29 := FALSE;
   Schlamm_AS.BEF_NHV.Bef.BF_Set_SW_chg := FALSE;
   Schlamm_AS.BEF_NHV.Bef.BF_Quit := FALSE;
   Schlamm_AS.BEF_NHV.SW_Hand := 0.0;

END_DATA_BLOCK

DATA_BLOCK "FB6_Kommunikation_IDB"
{ S7_Optimized_Access := 'TRUE' }
VERSION : 0.1
NON_RETAIN
"FB6_Kommunikation"

BEGIN

END_DATA_BLOCK

DATA_BLOCK "FB5_Automatik_Zulauf_Ablauf_IDB"
{ S7_Optimized_Access := 'TRUE' }
VERSION : 0.1
NON_RETAIN
"FB5_Automatik_Zulauf_Ablauf"

BEGIN

END_DATA_BLOCK

DATA_BLOCK "FB4_Automatik_Biocos_IDB"
{ S7_Optimized_Access := 'TRUE' }
VERSION : 0.1
NON_RETAIN
"FB4_Automatik_Biocos"

BEGIN

END_DATA_BLOCK

DATA_BLOCK "FB3_Automatik_Belebung_IDB"
{ S7_Optimized_Access := 'TRUE' }
VERSION : 0.1
NON_RETAIN
"FB3_Automatik_Belebung"

BEGIN

END_DATA_BLOCK

DATA_BLOCK "FB2_Messwerte_IDB"
{ S7_Optimized_Access := 'TRUE' }
VERSION : 0.1
NON_RETAIN
"FB2_Messwerte"

BEGIN

END_DATA_BLOCK

DATA_BLOCK "DB95_MWIdx"
{ S7_Optimized_Access := 'FALSE' }
VERSION : 0.1
NON_RETAIN
   STRUCT
      MaxIdx_ges : Int;
      MaxIdx : Array[0..6] of Byte;
      UV2ZEN : Array[0..6, 1..80] of Byte;
      ZEN2UV : Array[0..6, 1..132] of Byte;
   END_STRUCT;


BEGIN
   MaxIdx_ges := 17;
   MaxIdx[0] := 16#3E;
   MaxIdx[1] := 16#00;
   MaxIdx[2] := 16#00;
   MaxIdx[3] := 16#00;
   MaxIdx[4] := 16#00;
   MaxIdx[5] := 16#00;
   MaxIdx[6] := 16#26;
   UV2ZEN[0,1] := 16#01;
   UV2ZEN[0,2] := 16#02;
   UV2ZEN[0,3] := 16#03;
   UV2ZEN[0,4] := 16#04;
   UV2ZEN[0,5] := 16#05;
   UV2ZEN[0,6] := 16#06;
   UV2ZEN[0,7] := 16#07;
   UV2ZEN[0,8] := 16#08;
   UV2ZEN[0,9] := 16#09;
   UV2ZEN[0,10] := 16#0A;
   UV2ZEN[0,11] := 16#0B;
   UV2ZEN[0,12] := 16#0C;
   UV2ZEN[0,13] := 16#0D;
   UV2ZEN[0,14] := 16#0E;
   UV2ZEN[0,15] := 16#0F;
   UV2ZEN[0,16] := 16#10;
   UV2ZEN[0,17] := 16#11;
   UV2ZEN[0,18] := 16#12;
   UV2ZEN[0,19] := 16#13;
   UV2ZEN[0,20] := 16#14;
   UV2ZEN[0,21] := 16#15;
   UV2ZEN[0,22] := 16#16;
   UV2ZEN[0,23] := 16#17;
   UV2ZEN[0,24] := 16#18;
   UV2ZEN[0,25] := 16#19;
   UV2ZEN[0,26] := 16#1A;
   UV2ZEN[0,27] := 16#1B;
   UV2ZEN[0,28] := 16#1C;
   UV2ZEN[0,29] := 16#1D;
   UV2ZEN[0,30] := 16#1E;
   UV2ZEN[0,31] := 16#1F;
   UV2ZEN[0,32] := 16#20;
   UV2ZEN[0,33] := 16#21;
   UV2ZEN[0,34] := 16#22;
   UV2ZEN[0,35] := 16#23;
   UV2ZEN[0,36] := 16#24;
   UV2ZEN[0,37] := 16#25;
   UV2ZEN[0,38] := 16#26;
   UV2ZEN[0,39] := 16#27;
   UV2ZEN[0,40] := 16#28;
   UV2ZEN[0,41] := 16#00;
   UV2ZEN[0,42] := 16#00;
   UV2ZEN[0,43] := 16#00;
   UV2ZEN[0,44] := 16#2C;
   UV2ZEN[0,45] := 16#2D;
   UV2ZEN[0,46] := 16#2E;
   UV2ZEN[0,47] := 16#2F;
   UV2ZEN[0,48] := 16#30;
   UV2ZEN[0,49] := 16#31;
   UV2ZEN[0,50] := 16#32;
   UV2ZEN[0,51] := 16#33;
   UV2ZEN[0,52] := 16#34;
   UV2ZEN[0,53] := 16#35;
   UV2ZEN[0,54] := 16#36;
   UV2ZEN[0,55] := 16#37;
   UV2ZEN[0,56] := 16#38;
   UV2ZEN[0,57] := 16#39;
   UV2ZEN[0,58] := 16#3A;
   UV2ZEN[0,59] := 16#3B;
   UV2ZEN[0,60] := 16#3C;
   UV2ZEN[0,61] := 16#3D;
   UV2ZEN[0,62] := 16#3E;
   UV2ZEN[0,63] := 16#00;
   UV2ZEN[0,64] := 16#00;
   UV2ZEN[0,65] := 16#00;
   UV2ZEN[0,66] := 16#00;
   UV2ZEN[0,67] := 16#00;
   UV2ZEN[0,68] := 16#00;
   UV2ZEN[0,69] := 16#00;
   UV2ZEN[0,70] := 16#00;
   UV2ZEN[0,71] := 16#00;
   UV2ZEN[0,72] := 16#00;
   UV2ZEN[0,73] := 16#00;
   UV2ZEN[0,74] := 16#00;
   UV2ZEN[0,75] := 16#00;
   UV2ZEN[0,76] := 16#00;
   UV2ZEN[0,77] := 16#00;
   UV2ZEN[0,78] := 16#00;
   UV2ZEN[0,79] := 16#00;
   UV2ZEN[0,80] := 16#00;
   UV2ZEN[1,1] := 16#00;
   UV2ZEN[1,2] := 16#00;
   UV2ZEN[1,3] := 16#00;
   UV2ZEN[1,4] := 16#00;
   UV2ZEN[1,5] := 16#00;
   UV2ZEN[1,6] := 16#00;
   UV2ZEN[1,7] := 16#00;
   UV2ZEN[1,8] := 16#00;
   UV2ZEN[1,9] := 16#00;
   UV2ZEN[1,10] := 16#00;
   UV2ZEN[1,11] := 16#00;
   UV2ZEN[1,12] := 16#00;
   UV2ZEN[1,13] := 16#00;
   UV2ZEN[1,14] := 16#00;
   UV2ZEN[1,15] := 16#00;
   UV2ZEN[1,16] := 16#00;
   UV2ZEN[1,17] := 16#00;
   UV2ZEN[1,18] := 16#00;
   UV2ZEN[1,19] := 16#00;
   UV2ZEN[1,20] := 16#00;
   UV2ZEN[1,21] := 16#00;
   UV2ZEN[1,22] := 16#00;
   UV2ZEN[1,23] := 16#00;
   UV2ZEN[1,24] := 16#00;
   UV2ZEN[1,25] := 16#00;
   UV2ZEN[1,26] := 16#00;
   UV2ZEN[1,27] := 16#00;
   UV2ZEN[1,28] := 16#00;
   UV2ZEN[1,29] := 16#00;
   UV2ZEN[1,30] := 16#00;
   UV2ZEN[1,31] := 16#00;
   UV2ZEN[1,32] := 16#00;
   UV2ZEN[1,33] := 16#00;
   UV2ZEN[1,34] := 16#00;
   UV2ZEN[1,35] := 16#00;
   UV2ZEN[1,36] := 16#00;
   UV2ZEN[1,37] := 16#00;
   UV2ZEN[1,38] := 16#00;
   UV2ZEN[1,39] := 16#00;
   UV2ZEN[1,40] := 16#00;
   UV2ZEN[1,41] := 16#00;
   UV2ZEN[1,42] := 16#00;
   UV2ZEN[1,43] := 16#00;
   UV2ZEN[1,44] := 16#00;
   UV2ZEN[1,45] := 16#00;
   UV2ZEN[1,46] := 16#00;
   UV2ZEN[1,47] := 16#00;
   UV2ZEN[1,48] := 16#00;
   UV2ZEN[1,49] := 16#00;
   UV2ZEN[1,50] := 16#00;
   UV2ZEN[1,51] := 16#00;
   UV2ZEN[1,52] := 16#00;
   UV2ZEN[1,53] := 16#00;
   UV2ZEN[1,54] := 16#00;
   UV2ZEN[1,55] := 16#00;
   UV2ZEN[1,56] := 16#00;
   UV2ZEN[1,57] := 16#00;
   UV2ZEN[1,58] := 16#00;
   UV2ZEN[1,59] := 16#00;
   UV2ZEN[1,60] := 16#00;
   UV2ZEN[1,61] := 16#00;
   UV2ZEN[1,62] := 16#00;
   UV2ZEN[1,63] := 16#00;
   UV2ZEN[1,64] := 16#00;
   UV2ZEN[1,65] := 16#00;
   UV2ZEN[1,66] := 16#00;
   UV2ZEN[1,67] := 16#00;
   UV2ZEN[1,68] := 16#00;
   UV2ZEN[1,69] := 16#00;
   UV2ZEN[1,70] := 16#00;
   UV2ZEN[1,71] := 16#00;
   UV2ZEN[1,72] := 16#00;
   UV2ZEN[1,73] := 16#00;
   UV2ZEN[1,74] := 16#00;
   UV2ZEN[1,75] := 16#00;
   UV2ZEN[1,76] := 16#00;
   UV2ZEN[1,77] := 16#00;
   UV2ZEN[1,78] := 16#00;
   UV2ZEN[1,79] := 16#00;
   UV2ZEN[1,80] := 16#00;
   UV2ZEN[2,1] := 16#00;
   UV2ZEN[2,2] := 16#00;
   UV2ZEN[2,3] := 16#00;
   UV2ZEN[2,4] := 16#00;
   UV2ZEN[2,5] := 16#00;
   UV2ZEN[2,6] := 16#00;
   UV2ZEN[2,7] := 16#00;
   UV2ZEN[2,8] := 16#00;
   UV2ZEN[2,9] := 16#00;
   UV2ZEN[2,10] := 16#00;
   UV2ZEN[2,11] := 16#00;
   UV2ZEN[2,12] := 16#00;
   UV2ZEN[2,13] := 16#00;
   UV2ZEN[2,14] := 16#00;
   UV2ZEN[2,15] := 16#00;
   UV2ZEN[2,16] := 16#00;
   UV2ZEN[2,17] := 16#00;
   UV2ZEN[2,18] := 16#00;
   UV2ZEN[2,19] := 16#00;
   UV2ZEN[2,20] := 16#00;
   UV2ZEN[2,21] := 16#00;
   UV2ZEN[2,22] := 16#00;
   UV2ZEN[2,23] := 16#00;
   UV2ZEN[2,24] := 16#00;
   UV2ZEN[2,25] := 16#00;
   UV2ZEN[2,26] := 16#00;
   UV2ZEN[2,27] := 16#00;
   UV2ZEN[2,28] := 16#00;
   UV2ZEN[2,29] := 16#00;
   UV2ZEN[2,30] := 16#00;
   UV2ZEN[2,31] := 16#00;
   UV2ZEN[2,32] := 16#00;
   UV2ZEN[2,33] := 16#00;
   UV2ZEN[2,34] := 16#00;
   UV2ZEN[2,35] := 16#00;
   UV2ZEN[2,36] := 16#00;
   UV2ZEN[2,37] := 16#00;
   UV2ZEN[2,38] := 16#00;
   UV2ZEN[2,39] := 16#00;
   UV2ZEN[2,40] := 16#00;
   UV2ZEN[2,41] := 16#00;
   UV2ZEN[2,42] := 16#00;
   UV2ZEN[2,43] := 16#00;
   UV2ZEN[2,44] := 16#00;
   UV2ZEN[2,45] := 16#00;
   UV2ZEN[2,46] := 16#00;
   UV2ZEN[2,47] := 16#00;
   UV2ZEN[2,48] := 16#00;
   UV2ZEN[2,49] := 16#00;
   UV2ZEN[2,50] := 16#00;
   UV2ZEN[2,51] := 16#00;
   UV2ZEN[2,52] := 16#00;
   UV2ZEN[2,53] := 16#00;
   UV2ZEN[2,54] := 16#00;
   UV2ZEN[2,55] := 16#00;
   UV2ZEN[2,56] := 16#00;
   UV2ZEN[2,57] := 16#00;
   UV2ZEN[2,58] := 16#00;
   UV2ZEN[2,59] := 16#00;
   UV2ZEN[2,60] := 16#00;
   UV2ZEN[2,61] := 16#00;
   UV2ZEN[2,62] := 16#00;
   UV2ZEN[2,63] := 16#00;
   UV2ZEN[2,64] := 16#00;
   UV2ZEN[2,65] := 16#00;
   UV2ZEN[2,66] := 16#00;
   UV2ZEN[2,67] := 16#00;
   UV2ZEN[2,68] := 16#00;
   UV2ZEN[2,69] := 16#00;
   UV2ZEN[2,70] := 16#00;
   UV2ZEN[2,71] := 16#00;
   UV2ZEN[2,72] := 16#00;
   UV2ZEN[2,73] := 16#00;
   UV2ZEN[2,74] := 16#00;
   UV2ZEN[2,75] := 16#00;
   UV2ZEN[2,76] := 16#00;
   UV2ZEN[2,77] := 16#00;
   UV2ZEN[2,78] := 16#00;
   UV2ZEN[2,79] := 16#00;
   UV2ZEN[2,80] := 16#00;
   UV2ZEN[3,1] := 16#00;
   UV2ZEN[3,2] := 16#00;
   UV2ZEN[3,3] := 16#00;
   UV2ZEN[3,4] := 16#00;
   UV2ZEN[3,5] := 16#00;
   UV2ZEN[3,6] := 16#00;
   UV2ZEN[3,7] := 16#00;
   UV2ZEN[3,8] := 16#00;
   UV2ZEN[3,9] := 16#00;
   UV2ZEN[3,10] := 16#00;
   UV2ZEN[3,11] := 16#00;
   UV2ZEN[3,12] := 16#00;
   UV2ZEN[3,13] := 16#00;
   UV2ZEN[3,14] := 16#00;
   UV2ZEN[3,15] := 16#00;
   UV2ZEN[3,16] := 16#00;
   UV2ZEN[3,17] := 16#00;
   UV2ZEN[3,18] := 16#00;
   UV2ZEN[3,19] := 16#00;
   UV2ZEN[3,20] := 16#00;
   UV2ZEN[3,21] := 16#00;
   UV2ZEN[3,22] := 16#00;
   UV2ZEN[3,23] := 16#00;
   UV2ZEN[3,24] := 16#00;
   UV2ZEN[3,25] := 16#00;
   UV2ZEN[3,26] := 16#00;
   UV2ZEN[3,27] := 16#00;
   UV2ZEN[3,28] := 16#00;
   UV2ZEN[3,29] := 16#00;
   UV2ZEN[3,30] := 16#00;
   UV2ZEN[3,31] := 16#00;
   UV2ZEN[3,32] := 16#00;
   UV2ZEN[3,33] := 16#00;
   UV2ZEN[3,34] := 16#00;
   UV2ZEN[3,35] := 16#00;
   UV2ZEN[3,36] := 16#00;
   UV2ZEN[3,37] := 16#00;
   UV2ZEN[3,38] := 16#00;
   UV2ZEN[3,39] := 16#00;
   UV2ZEN[3,40] := 16#00;
   UV2ZEN[3,41] := 16#00;
   UV2ZEN[3,42] := 16#00;
   UV2ZEN[3,43] := 16#00;
   UV2ZEN[3,44] := 16#00;
   UV2ZEN[3,45] := 16#00;
   UV2ZEN[3,46] := 16#00;
   UV2ZEN[3,47] := 16#00;
   UV2ZEN[3,48] := 16#00;
   UV2ZEN[3,49] := 16#00;
   UV2ZEN[3,50] := 16#00;
   UV2ZEN[3,51] := 16#00;
   UV2ZEN[3,52] := 16#00;
   UV2ZEN[3,53] := 16#00;
   UV2ZEN[3,54] := 16#00;
   UV2ZEN[3,55] := 16#00;
   UV2ZEN[3,56] := 16#00;
   UV2ZEN[3,57] := 16#00;
   UV2ZEN[3,58] := 16#00;
   UV2ZEN[3,59] := 16#00;
   UV2ZEN[3,60] := 16#00;
   UV2ZEN[3,61] := 16#00;
   UV2ZEN[3,62] := 16#00;
   UV2ZEN[3,63] := 16#00;
   UV2ZEN[3,64] := 16#00;
   UV2ZEN[3,65] := 16#00;
   UV2ZEN[3,66] := 16#00;
   UV2ZEN[3,67] := 16#00;
   UV2ZEN[3,68] := 16#00;
   UV2ZEN[3,69] := 16#00;
   UV2ZEN[3,70] := 16#00;
   UV2ZEN[3,71] := 16#00;
   UV2ZEN[3,72] := 16#00;
   UV2ZEN[3,73] := 16#00;
   UV2ZEN[3,74] := 16#00;
   UV2ZEN[3,75] := 16#00;
   UV2ZEN[3,76] := 16#00;
   UV2ZEN[3,77] := 16#00;
   UV2ZEN[3,78] := 16#00;
   UV2ZEN[3,79] := 16#00;
   UV2ZEN[3,80] := 16#00;
   UV2ZEN[4,1] := 16#00;
   UV2ZEN[4,2] := 16#00;
   UV2ZEN[4,3] := 16#00;
   UV2ZEN[4,4] := 16#00;
   UV2ZEN[4,5] := 16#00;
   UV2ZEN[4,6] := 16#00;
   UV2ZEN[4,7] := 16#00;
   UV2ZEN[4,8] := 16#00;
   UV2ZEN[4,9] := 16#00;
   UV2ZEN[4,10] := 16#00;
   UV2ZEN[4,11] := 16#00;
   UV2ZEN[4,12] := 16#00;
   UV2ZEN[4,13] := 16#00;
   UV2ZEN[4,14] := 16#00;
   UV2ZEN[4,15] := 16#00;
   UV2ZEN[4,16] := 16#00;
   UV2ZEN[4,17] := 16#00;
   UV2ZEN[4,18] := 16#00;
   UV2ZEN[4,19] := 16#00;
   UV2ZEN[4,20] := 16#00;
   UV2ZEN[4,21] := 16#00;
   UV2ZEN[4,22] := 16#00;
   UV2ZEN[4,23] := 16#00;
   UV2ZEN[4,24] := 16#00;
   UV2ZEN[4,25] := 16#00;
   UV2ZEN[4,26] := 16#00;
   UV2ZEN[4,27] := 16#00;
   UV2ZEN[4,28] := 16#00;
   UV2ZEN[4,29] := 16#00;
   UV2ZEN[4,30] := 16#00;
   UV2ZEN[4,31] := 16#00;
   UV2ZEN[4,32] := 16#00;
   UV2ZEN[4,33] := 16#00;
   UV2ZEN[4,34] := 16#00;
   UV2ZEN[4,35] := 16#00;
   UV2ZEN[4,36] := 16#00;
   UV2ZEN[4,37] := 16#00;
   UV2ZEN[4,38] := 16#00;
   UV2ZEN[4,39] := 16#00;
   UV2ZEN[4,40] := 16#00;
   UV2ZEN[4,41] := 16#00;
   UV2ZEN[4,42] := 16#00;
   UV2ZEN[4,43] := 16#00;
   UV2ZEN[4,44] := 16#00;
   UV2ZEN[4,45] := 16#00;
   UV2ZEN[4,46] := 16#00;
   UV2ZEN[4,47] := 16#00;
   UV2ZEN[4,48] := 16#00;
   UV2ZEN[4,49] := 16#00;
   UV2ZEN[4,50] := 16#00;
   UV2ZEN[4,51] := 16#00;
   UV2ZEN[4,52] := 16#00;
   UV2ZEN[4,53] := 16#00;
   UV2ZEN[4,54] := 16#00;
   UV2ZEN[4,55] := 16#00;
   UV2ZEN[4,56] := 16#00;
   UV2ZEN[4,57] := 16#00;
   UV2ZEN[4,58] := 16#00;
   UV2ZEN[4,59] := 16#00;
   UV2ZEN[4,60] := 16#00;
   UV2ZEN[4,61] := 16#00;
   UV2ZEN[4,62] := 16#00;
   UV2ZEN[4,63] := 16#00;
   UV2ZEN[4,64] := 16#00;
   UV2ZEN[4,65] := 16#00;
   UV2ZEN[4,66] := 16#00;
   UV2ZEN[4,67] := 16#00;
   UV2ZEN[4,68] := 16#00;
   UV2ZEN[4,69] := 16#00;
   UV2ZEN[4,70] := 16#00;
   UV2ZEN[4,71] := 16#00;
   UV2ZEN[4,72] := 16#00;
   UV2ZEN[4,73] := 16#00;
   UV2ZEN[4,74] := 16#00;
   UV2ZEN[4,75] := 16#00;
   UV2ZEN[4,76] := 16#00;
   UV2ZEN[4,77] := 16#00;
   UV2ZEN[4,78] := 16#00;
   UV2ZEN[4,79] := 16#00;
   UV2ZEN[4,80] := 16#00;
   UV2ZEN[5,1] := 16#00;
   UV2ZEN[5,2] := 16#00;
   UV2ZEN[5,3] := 16#00;
   UV2ZEN[5,4] := 16#00;
   UV2ZEN[5,5] := 16#00;
   UV2ZEN[5,6] := 16#00;
   UV2ZEN[5,7] := 16#00;
   UV2ZEN[5,8] := 16#00;
   UV2ZEN[5,9] := 16#00;
   UV2ZEN[5,10] := 16#00;
   UV2ZEN[5,11] := 16#00;
   UV2ZEN[5,12] := 16#00;
   UV2ZEN[5,13] := 16#00;
   UV2ZEN[5,14] := 16#00;
   UV2ZEN[5,15] := 16#00;
   UV2ZEN[5,16] := 16#00;
   UV2ZEN[5,17] := 16#00;
   UV2ZEN[5,18] := 16#00;
   UV2ZEN[5,19] := 16#00;
   UV2ZEN[5,20] := 16#00;
   UV2ZEN[5,21] := 16#00;
   UV2ZEN[5,22] := 16#00;
   UV2ZEN[5,23] := 16#00;
   UV2ZEN[5,24] := 16#00;
   UV2ZEN[5,25] := 16#00;
   UV2ZEN[5,26] := 16#00;
   UV2ZEN[5,27] := 16#00;
   UV2ZEN[5,28] := 16#00;
   UV2ZEN[5,29] := 16#00;
   UV2ZEN[5,30] := 16#00;
   UV2ZEN[5,31] := 16#00;
   UV2ZEN[5,32] := 16#00;
   UV2ZEN[5,33] := 16#00;
   UV2ZEN[5,34] := 16#00;
   UV2ZEN[5,35] := 16#00;
   UV2ZEN[5,36] := 16#00;
   UV2ZEN[5,37] := 16#00;
   UV2ZEN[5,38] := 16#00;
   UV2ZEN[5,39] := 16#00;
   UV2ZEN[5,40] := 16#00;
   UV2ZEN[5,41] := 16#00;
   UV2ZEN[5,42] := 16#00;
   UV2ZEN[5,43] := 16#00;
   UV2ZEN[5,44] := 16#00;
   UV2ZEN[5,45] := 16#00;
   UV2ZEN[5,46] := 16#00;
   UV2ZEN[5,47] := 16#00;
   UV2ZEN[5,48] := 16#00;
   UV2ZEN[5,49] := 16#00;
   UV2ZEN[5,50] := 16#00;
   UV2ZEN[5,51] := 16#00;
   UV2ZEN[5,52] := 16#00;
   UV2ZEN[5,53] := 16#00;
   UV2ZEN[5,54] := 16#00;
   UV2ZEN[5,55] := 16#00;
   UV2ZEN[5,56] := 16#00;
   UV2ZEN[5,57] := 16#00;
   UV2ZEN[5,58] := 16#00;
   UV2ZEN[5,59] := 16#00;
   UV2ZEN[5,60] := 16#00;
   UV2ZEN[5,61] := 16#00;
   UV2ZEN[5,62] := 16#00;
   UV2ZEN[5,63] := 16#00;
   UV2ZEN[5,64] := 16#00;
   UV2ZEN[5,65] := 16#00;
   UV2ZEN[5,66] := 16#00;
   UV2ZEN[5,67] := 16#00;
   UV2ZEN[5,68] := 16#00;
   UV2ZEN[5,69] := 16#00;
   UV2ZEN[5,70] := 16#00;
   UV2ZEN[5,71] := 16#00;
   UV2ZEN[5,72] := 16#00;
   UV2ZEN[5,73] := 16#00;
   UV2ZEN[5,74] := 16#00;
   UV2ZEN[5,75] := 16#00;
   UV2ZEN[5,76] := 16#00;
   UV2ZEN[5,77] := 16#00;
   UV2ZEN[5,78] := 16#00;
   UV2ZEN[5,79] := 16#00;
   UV2ZEN[5,80] := 16#00;
   UV2ZEN[6,1] := 16#29;
   UV2ZEN[6,2] := 16#2A;
   UV2ZEN[6,3] := 16#2B;
   UV2ZEN[6,4] := 16#3F;
   UV2ZEN[6,5] := 16#40;
   UV2ZEN[6,6] := 16#41;
   UV2ZEN[6,7] := 16#42;
   UV2ZEN[6,8] := 16#43;
   UV2ZEN[6,9] := 16#44;
   UV2ZEN[6,10] := 16#45;
   UV2ZEN[6,11] := 16#46;
   UV2ZEN[6,12] := 16#47;
   UV2ZEN[6,13] := 16#48;
   UV2ZEN[6,14] := 16#49;
   UV2ZEN[6,15] := 16#4A;
   UV2ZEN[6,16] := 16#4B;
   UV2ZEN[6,17] := 16#4C;
   UV2ZEN[6,18] := 16#4D;
   UV2ZEN[6,19] := 16#4E;
   UV2ZEN[6,20] := 16#4F;
   UV2ZEN[6,21] := 16#50;
   UV2ZEN[6,22] := 16#51;
   UV2ZEN[6,23] := 16#52;
   UV2ZEN[6,24] := 16#53;
   UV2ZEN[6,25] := 16#54;
   UV2ZEN[6,26] := 16#55;
   UV2ZEN[6,27] := 16#56;
   UV2ZEN[6,28] := 16#57;
   UV2ZEN[6,29] := 16#58;
   UV2ZEN[6,30] := 16#59;
   UV2ZEN[6,31] := 16#5A;
   UV2ZEN[6,32] := 16#5B;
   UV2ZEN[6,33] := 16#5C;
   UV2ZEN[6,34] := 16#5D;
   UV2ZEN[6,35] := 16#5E;
   UV2ZEN[6,36] := 16#5F;
   UV2ZEN[6,37] := 16#60;
   UV2ZEN[6,38] := 16#61;
   UV2ZEN[6,39] := 16#00;
   UV2ZEN[6,40] := 16#00;
   UV2ZEN[6,41] := 16#00;
   UV2ZEN[6,42] := 16#00;
   UV2ZEN[6,43] := 16#00;
   UV2ZEN[6,44] := 16#00;
   UV2ZEN[6,45] := 16#00;
   UV2ZEN[6,46] := 16#00;
   UV2ZEN[6,47] := 16#00;
   UV2ZEN[6,48] := 16#00;
   UV2ZEN[6,49] := 16#00;
   UV2ZEN[6,50] := 16#00;
   UV2ZEN[6,51] := 16#00;
   UV2ZEN[6,52] := 16#00;
   UV2ZEN[6,53] := 16#00;
   UV2ZEN[6,54] := 16#00;
   UV2ZEN[6,55] := 16#00;
   UV2ZEN[6,56] := 16#00;
   UV2ZEN[6,57] := 16#00;
   UV2ZEN[6,58] := 16#00;
   UV2ZEN[6,59] := 16#00;
   UV2ZEN[6,60] := 16#00;
   UV2ZEN[6,61] := 16#00;
   UV2ZEN[6,62] := 16#00;
   UV2ZEN[6,63] := 16#00;
   UV2ZEN[6,64] := 16#00;
   UV2ZEN[6,65] := 16#00;
   UV2ZEN[6,66] := 16#00;
   UV2ZEN[6,67] := 16#00;
   UV2ZEN[6,68] := 16#00;
   UV2ZEN[6,69] := 16#00;
   UV2ZEN[6,70] := 16#00;
   UV2ZEN[6,71] := 16#00;
   UV2ZEN[6,72] := 16#00;
   UV2ZEN[6,73] := 16#00;
   UV2ZEN[6,74] := 16#00;
   UV2ZEN[6,75] := 16#00;
   UV2ZEN[6,76] := 16#00;
   UV2ZEN[6,77] := 16#00;
   UV2ZEN[6,78] := 16#00;
   UV2ZEN[6,79] := 16#00;
   UV2ZEN[6,80] := 16#00;
   ZEN2UV[0,1] := 16#01;
   ZEN2UV[0,2] := 16#02;
   ZEN2UV[0,3] := 16#03;
   ZEN2UV[0,4] := 16#04;
   ZEN2UV[0,5] := 16#05;
   ZEN2UV[0,6] := 16#06;
   ZEN2UV[0,7] := 16#07;
   ZEN2UV[0,8] := 16#08;
   ZEN2UV[0,9] := 16#09;
   ZEN2UV[0,10] := 16#0A;
   ZEN2UV[0,11] := 16#0B;
   ZEN2UV[0,12] := 16#0C;
   ZEN2UV[0,13] := 16#0D;
   ZEN2UV[0,14] := 16#0E;
   ZEN2UV[0,15] := 16#0F;
   ZEN2UV[0,16] := 16#10;
   ZEN2UV[0,17] := 16#11;
   ZEN2UV[0,18] := 16#12;
   ZEN2UV[0,19] := 16#13;
   ZEN2UV[0,20] := 16#14;
   ZEN2UV[0,21] := 16#15;
   ZEN2UV[0,22] := 16#16;
   ZEN2UV[0,23] := 16#17;
   ZEN2UV[0,24] := 16#18;
   ZEN2UV[0,25] := 16#19;
   ZEN2UV[0,26] := 16#1A;
   ZEN2UV[0,27] := 16#1B;
   ZEN2UV[0,28] := 16#1C;
   ZEN2UV[0,29] := 16#1D;
   ZEN2UV[0,30] := 16#1E;
   ZEN2UV[0,31] := 16#1F;
   ZEN2UV[0,32] := 16#20;
   ZEN2UV[0,33] := 16#21;
   ZEN2UV[0,34] := 16#22;
   ZEN2UV[0,35] := 16#23;
   ZEN2UV[0,36] := 16#24;
   ZEN2UV[0,37] := 16#25;
   ZEN2UV[0,38] := 16#26;
   ZEN2UV[0,39] := 16#27;
   ZEN2UV[0,40] := 16#28;
   ZEN2UV[0,41] := 16#00;
   ZEN2UV[0,42] := 16#00;
   ZEN2UV[0,43] := 16#00;
   ZEN2UV[0,44] := 16#2C;
   ZEN2UV[0,45] := 16#2D;
   ZEN2UV[0,46] := 16#2E;
   ZEN2UV[0,47] := 16#2F;
   ZEN2UV[0,48] := 16#30;
   ZEN2UV[0,49] := 16#31;
   ZEN2UV[0,50] := 16#32;
   ZEN2UV[0,51] := 16#33;
   ZEN2UV[0,52] := 16#34;
   ZEN2UV[0,53] := 16#35;
   ZEN2UV[0,54] := 16#36;
   ZEN2UV[0,55] := 16#37;
   ZEN2UV[0,56] := 16#38;
   ZEN2UV[0,57] := 16#39;
   ZEN2UV[0,58] := 16#3A;
   ZEN2UV[0,59] := 16#3B;
   ZEN2UV[0,60] := 16#3C;
   ZEN2UV[0,61] := 16#3D;
   ZEN2UV[0,62] := 16#3E;
   ZEN2UV[0,63] := 16#00;
   ZEN2UV[0,64] := 16#00;
   ZEN2UV[0,65] := 16#00;
   ZEN2UV[0,66] := 16#00;
   ZEN2UV[0,67] := 16#00;
   ZEN2UV[0,68] := 16#00;
   ZEN2UV[0,69] := 16#00;
   ZEN2UV[0,70] := 16#00;
   ZEN2UV[0,71] := 16#00;
   ZEN2UV[0,72] := 16#00;
   ZEN2UV[0,73] := 16#00;
   ZEN2UV[0,74] := 16#00;
   ZEN2UV[0,75] := 16#00;
   ZEN2UV[0,76] := 16#00;
   ZEN2UV[0,77] := 16#00;
   ZEN2UV[0,78] := 16#00;
   ZEN2UV[0,79] := 16#00;
   ZEN2UV[0,80] := 16#00;
   ZEN2UV[0,81] := 16#00;
   ZEN2UV[0,82] := 16#00;
   ZEN2UV[0,83] := 16#00;
   ZEN2UV[0,84] := 16#00;
   ZEN2UV[0,85] := 16#00;
   ZEN2UV[0,86] := 16#00;
   ZEN2UV[0,87] := 16#00;
   ZEN2UV[0,88] := 16#00;
   ZEN2UV[0,89] := 16#00;
   ZEN2UV[0,90] := 16#00;
   ZEN2UV[0,91] := 16#00;
   ZEN2UV[0,92] := 16#00;
   ZEN2UV[0,93] := 16#00;
   ZEN2UV[0,94] := 16#00;
   ZEN2UV[0,95] := 16#00;
   ZEN2UV[0,96] := 16#00;
   ZEN2UV[0,97] := 16#00;
   ZEN2UV[0,98] := 16#00;
   ZEN2UV[0,99] := 16#00;
   ZEN2UV[0,100] := 16#00;
   ZEN2UV[0,101] := 16#00;
   ZEN2UV[0,102] := 16#00;
   ZEN2UV[0,103] := 16#00;
   ZEN2UV[0,104] := 16#00;
   ZEN2UV[0,105] := 16#00;
   ZEN2UV[0,106] := 16#00;
   ZEN2UV[0,107] := 16#00;
   ZEN2UV[0,108] := 16#00;
   ZEN2UV[0,109] := 16#00;
   ZEN2UV[0,110] := 16#00;
   ZEN2UV[0,111] := 16#00;
   ZEN2UV[0,112] := 16#00;
   ZEN2UV[0,113] := 16#00;
   ZEN2UV[0,114] := 16#00;
   ZEN2UV[0,115] := 16#00;
   ZEN2UV[0,116] := 16#00;
   ZEN2UV[0,117] := 16#00;
   ZEN2UV[0,118] := 16#00;
   ZEN2UV[0,119] := 16#00;
   ZEN2UV[0,120] := 16#00;
   ZEN2UV[0,121] := 16#00;
   ZEN2UV[0,122] := 16#00;
   ZEN2UV[0,123] := 16#00;
   ZEN2UV[0,124] := 16#00;
   ZEN2UV[0,125] := 16#00;
   ZEN2UV[0,126] := 16#00;
   ZEN2UV[0,127] := 16#00;
   ZEN2UV[0,128] := 16#00;
   ZEN2UV[0,129] := 16#00;
   ZEN2UV[0,130] := 16#00;
   ZEN2UV[0,131] := 16#00;
   ZEN2UV[0,132] := 16#00;
   ZEN2UV[1,1] := 16#00;
   ZEN2UV[1,2] := 16#00;
   ZEN2UV[1,3] := 16#00;
   ZEN2UV[1,4] := 16#00;
   ZEN2UV[1,5] := 16#00;
   ZEN2UV[1,6] := 16#00;
   ZEN2UV[1,7] := 16#00;
   ZEN2UV[1,8] := 16#00;
   ZEN2UV[1,9] := 16#00;
   ZEN2UV[1,10] := 16#00;
   ZEN2UV[1,11] := 16#00;
   ZEN2UV[1,12] := 16#00;
   ZEN2UV[1,13] := 16#00;
   ZEN2UV[1,14] := 16#00;
   ZEN2UV[1,15] := 16#00;
   ZEN2UV[1,16] := 16#00;
   ZEN2UV[1,17] := 16#00;
   ZEN2UV[1,18] := 16#00;
   ZEN2UV[1,19] := 16#00;
   ZEN2UV[1,20] := 16#00;
   ZEN2UV[1,21] := 16#00;
   ZEN2UV[1,22] := 16#00;
   ZEN2UV[1,23] := 16#00;
   ZEN2UV[1,24] := 16#00;
   ZEN2UV[1,25] := 16#00;
   ZEN2UV[1,26] := 16#00;
   ZEN2UV[1,27] := 16#00;
   ZEN2UV[1,28] := 16#00;
   ZEN2UV[1,29] := 16#00;
   ZEN2UV[1,30] := 16#00;
   ZEN2UV[1,31] := 16#00;
   ZEN2UV[1,32] := 16#00;
   ZEN2UV[1,33] := 16#00;
   ZEN2UV[1,34] := 16#00;
   ZEN2UV[1,35] := 16#00;
   ZEN2UV[1,36] := 16#00;
   ZEN2UV[1,37] := 16#00;
   ZEN2UV[1,38] := 16#00;
   ZEN2UV[1,39] := 16#00;
   ZEN2UV[1,40] := 16#00;
   ZEN2UV[1,41] := 16#00;
   ZEN2UV[1,42] := 16#00;
   ZEN2UV[1,43] := 16#00;
   ZEN2UV[1,44] := 16#00;
   ZEN2UV[1,45] := 16#00;
   ZEN2UV[1,46] := 16#00;
   ZEN2UV[1,47] := 16#00;
   ZEN2UV[1,48] := 16#00;
   ZEN2UV[1,49] := 16#00;
   ZEN2UV[1,50] := 16#00;
   ZEN2UV[1,51] := 16#00;
   ZEN2UV[1,52] := 16#00;
   ZEN2UV[1,53] := 16#00;
   ZEN2UV[1,54] := 16#00;
   ZEN2UV[1,55] := 16#00;
   ZEN2UV[1,56] := 16#00;
   ZEN2UV[1,57] := 16#00;
   ZEN2UV[1,58] := 16#00;
   ZEN2UV[1,59] := 16#00;
   ZEN2UV[1,60] := 16#00;
   ZEN2UV[1,61] := 16#00;
   ZEN2UV[1,62] := 16#00;
   ZEN2UV[1,63] := 16#00;
   ZEN2UV[1,64] := 16#00;
   ZEN2UV[1,65] := 16#00;
   ZEN2UV[1,66] := 16#00;
   ZEN2UV[1,67] := 16#00;
   ZEN2UV[1,68] := 16#00;
   ZEN2UV[1,69] := 16#00;
   ZEN2UV[1,70] := 16#00;
   ZEN2UV[1,71] := 16#00;
   ZEN2UV[1,72] := 16#00;
   ZEN2UV[1,73] := 16#00;
   ZEN2UV[1,74] := 16#00;
   ZEN2UV[1,75] := 16#00;
   ZEN2UV[1,76] := 16#00;
   ZEN2UV[1,77] := 16#00;
   ZEN2UV[1,78] := 16#00;
   ZEN2UV[1,79] := 16#00;
   ZEN2UV[1,80] := 16#00;
   ZEN2UV[1,81] := 16#00;
   ZEN2UV[1,82] := 16#00;
   ZEN2UV[1,83] := 16#00;
   ZEN2UV[1,84] := 16#00;
   ZEN2UV[1,85] := 16#00;
   ZEN2UV[1,86] := 16#00;
   ZEN2UV[1,87] := 16#00;
   ZEN2UV[1,88] := 16#00;
   ZEN2UV[1,89] := 16#00;
   ZEN2UV[1,90] := 16#00;
   ZEN2UV[1,91] := 16#00;
   ZEN2UV[1,92] := 16#00;
   ZEN2UV[1,93] := 16#00;
   ZEN2UV[1,94] := 16#00;
   ZEN2UV[1,95] := 16#00;
   ZEN2UV[1,96] := 16#00;
   ZEN2UV[1,97] := 16#00;
   ZEN2UV[1,98] := 16#00;
   ZEN2UV[1,99] := 16#00;
   ZEN2UV[1,100] := 16#00;
   ZEN2UV[1,101] := 16#00;
   ZEN2UV[1,102] := 16#00;
   ZEN2UV[1,103] := 16#00;
   ZEN2UV[1,104] := 16#00;
   ZEN2UV[1,105] := 16#00;
   ZEN2UV[1,106] := 16#00;
   ZEN2UV[1,107] := 16#00;
   ZEN2UV[1,108] := 16#00;
   ZEN2UV[1,109] := 16#00;
   ZEN2UV[1,110] := 16#00;
   ZEN2UV[1,111] := 16#00;
   ZEN2UV[1,112] := 16#00;
   ZEN2UV[1,113] := 16#00;
   ZEN2UV[1,114] := 16#00;
   ZEN2UV[1,115] := 16#00;
   ZEN2UV[1,116] := 16#00;
   ZEN2UV[1,117] := 16#00;
   ZEN2UV[1,118] := 16#00;
   ZEN2UV[1,119] := 16#00;
   ZEN2UV[1,120] := 16#00;
   ZEN2UV[1,121] := 16#00;
   ZEN2UV[1,122] := 16#00;
   ZEN2UV[1,123] := 16#00;
   ZEN2UV[1,124] := 16#00;
   ZEN2UV[1,125] := 16#00;
   ZEN2UV[1,126] := 16#00;
   ZEN2UV[1,127] := 16#00;
   ZEN2UV[1,128] := 16#00;
   ZEN2UV[1,129] := 16#00;
   ZEN2UV[1,130] := 16#00;
   ZEN2UV[1,131] := 16#00;
   ZEN2UV[1,132] := 16#00;
   ZEN2UV[2,1] := 16#00;
   ZEN2UV[2,2] := 16#00;
   ZEN2UV[2,3] := 16#00;
   ZEN2UV[2,4] := 16#00;
   ZEN2UV[2,5] := 16#00;
   ZEN2UV[2,6] := 16#00;
   ZEN2UV[2,7] := 16#00;
   ZEN2UV[2,8] := 16#00;
   ZEN2UV[2,9] := 16#00;
   ZEN2UV[2,10] := 16#00;
   ZEN2UV[2,11] := 16#00;
   ZEN2UV[2,12] := 16#00;
   ZEN2UV[2,13] := 16#00;
   ZEN2UV[2,14] := 16#00;
   ZEN2UV[2,15] := 16#00;
   ZEN2UV[2,16] := 16#00;
   ZEN2UV[2,17] := 16#00;
   ZEN2UV[2,18] := 16#00;
   ZEN2UV[2,19] := 16#00;
   ZEN2UV[2,20] := 16#00;
   ZEN2UV[2,21] := 16#00;
   ZEN2UV[2,22] := 16#00;
   ZEN2UV[2,23] := 16#00;
   ZEN2UV[2,24] := 16#00;
   ZEN2UV[2,25] := 16#00;
   ZEN2UV[2,26] := 16#00;
   ZEN2UV[2,27] := 16#00;
   ZEN2UV[2,28] := 16#00;
   ZEN2UV[2,29] := 16#00;
   ZEN2UV[2,30] := 16#00;
   ZEN2UV[2,31] := 16#00;
   ZEN2UV[2,32] := 16#00;
   ZEN2UV[2,33] := 16#00;
   ZEN2UV[2,34] := 16#00;
   ZEN2UV[2,35] := 16#00;
   ZEN2UV[2,36] := 16#00;
   ZEN2UV[2,37] := 16#00;
   ZEN2UV[2,38] := 16#00;
   ZEN2UV[2,39] := 16#00;
   ZEN2UV[2,40] := 16#00;
   ZEN2UV[2,41] := 16#00;
   ZEN2UV[2,42] := 16#00;
   ZEN2UV[2,43] := 16#00;
   ZEN2UV[2,44] := 16#00;
   ZEN2UV[2,45] := 16#00;
   ZEN2UV[2,46] := 16#00;
   ZEN2UV[2,47] := 16#00;
   ZEN2UV[2,48] := 16#00;
   ZEN2UV[2,49] := 16#00;
   ZEN2UV[2,50] := 16#00;
   ZEN2UV[2,51] := 16#00;
   ZEN2UV[2,52] := 16#00;
   ZEN2UV[2,53] := 16#00;
   ZEN2UV[2,54] := 16#00;
   ZEN2UV[2,55] := 16#00;
   ZEN2UV[2,56] := 16#00;
   ZEN2UV[2,57] := 16#00;
   ZEN2UV[2,58] := 16#00;
   ZEN2UV[2,59] := 16#00;
   ZEN2UV[2,60] := 16#00;
   ZEN2UV[2,61] := 16#00;
   ZEN2UV[2,62] := 16#00;
   ZEN2UV[2,63] := 16#00;
   ZEN2UV[2,64] := 16#00;
   ZEN2UV[2,65] := 16#00;
   ZEN2UV[2,66] := 16#00;
   ZEN2UV[2,67] := 16#00;
   ZEN2UV[2,68] := 16#00;
   ZEN2UV[2,69] := 16#00;
   ZEN2UV[2,70] := 16#00;
   ZEN2UV[2,71] := 16#00;
   ZEN2UV[2,72] := 16#00;
   ZEN2UV[2,73] := 16#00;
   ZEN2UV[2,74] := 16#00;
   ZEN2UV[2,75] := 16#00;
   ZEN2UV[2,76] := 16#00;
   ZEN2UV[2,77] := 16#00;
   ZEN2UV[2,78] := 16#00;
   ZEN2UV[2,79] := 16#00;
   ZEN2UV[2,80] := 16#00;
   ZEN2UV[2,81] := 16#00;
   ZEN2UV[2,82] := 16#00;
   ZEN2UV[2,83] := 16#00;
   ZEN2UV[2,84] := 16#00;
   ZEN2UV[2,85] := 16#00;
   ZEN2UV[2,86] := 16#00;
   ZEN2UV[2,87] := 16#00;
   ZEN2UV[2,88] := 16#00;
   ZEN2UV[2,89] := 16#00;
   ZEN2UV[2,90] := 16#00;
   ZEN2UV[2,91] := 16#00;
   ZEN2UV[2,92] := 16#00;
   ZEN2UV[2,93] := 16#00;
   ZEN2UV[2,94] := 16#00;
   ZEN2UV[2,95] := 16#00;
   ZEN2UV[2,96] := 16#00;
   ZEN2UV[2,97] := 16#00;
   ZEN2UV[2,98] := 16#00;
   ZEN2UV[2,99] := 16#00;
   ZEN2UV[2,100] := 16#00;
   ZEN2UV[2,101] := 16#00;
   ZEN2UV[2,102] := 16#00;
   ZEN2UV[2,103] := 16#00;
   ZEN2UV[2,104] := 16#00;
   ZEN2UV[2,105] := 16#00;
   ZEN2UV[2,106] := 16#00;
   ZEN2UV[2,107] := 16#00;
   ZEN2UV[2,108] := 16#00;
   ZEN2UV[2,109] := 16#00;
   ZEN2UV[2,110] := 16#00;
   ZEN2UV[2,111] := 16#00;
   ZEN2UV[2,112] := 16#00;
   ZEN2UV[2,113] := 16#00;
   ZEN2UV[2,114] := 16#00;
   ZEN2UV[2,115] := 16#00;
   ZEN2UV[2,116] := 16#00;
   ZEN2UV[2,117] := 16#00;
   ZEN2UV[2,118] := 16#00;
   ZEN2UV[2,119] := 16#00;
   ZEN2UV[2,120] := 16#00;
   ZEN2UV[2,121] := 16#00;
   ZEN2UV[2,122] := 16#00;
   ZEN2UV[2,123] := 16#00;
   ZEN2UV[2,124] := 16#00;
   ZEN2UV[2,125] := 16#00;
   ZEN2UV[2,126] := 16#00;
   ZEN2UV[2,127] := 16#00;
   ZEN2UV[2,128] := 16#00;
   ZEN2UV[2,129] := 16#00;
   ZEN2UV[2,130] := 16#00;
   ZEN2UV[2,131] := 16#00;
   ZEN2UV[2,132] := 16#00;
   ZEN2UV[3,1] := 16#00;
   ZEN2UV[3,2] := 16#00;
   ZEN2UV[3,3] := 16#00;
   ZEN2UV[3,4] := 16#00;
   ZEN2UV[3,5] := 16#00;
   ZEN2UV[3,6] := 16#00;
   ZEN2UV[3,7] := 16#00;
   ZEN2UV[3,8] := 16#00;
   ZEN2UV[3,9] := 16#00;
   ZEN2UV[3,10] := 16#00;
   ZEN2UV[3,11] := 16#00;
   ZEN2UV[3,12] := 16#00;
   ZEN2UV[3,13] := 16#00;
   ZEN2UV[3,14] := 16#00;
   ZEN2UV[3,15] := 16#00;
   ZEN2UV[3,16] := 16#00;
   ZEN2UV[3,17] := 16#00;
   ZEN2UV[3,18] := 16#00;
   ZEN2UV[3,19] := 16#00;
   ZEN2UV[3,20] := 16#00;
   ZEN2UV[3,21] := 16#00;
   ZEN2UV[3,22] := 16#00;
   ZEN2UV[3,23] := 16#00;
   ZEN2UV[3,24] := 16#00;
   ZEN2UV[3,25] := 16#00;
   ZEN2UV[3,26] := 16#00;
   ZEN2UV[3,27] := 16#00;
   ZEN2UV[3,28] := 16#00;
   ZEN2UV[3,29] := 16#00;
   ZEN2UV[3,30] := 16#00;
   ZEN2UV[3,31] := 16#00;
   ZEN2UV[3,32] := 16#00;
   ZEN2UV[3,33] := 16#00;
   ZEN2UV[3,34] := 16#00;
   ZEN2UV[3,35] := 16#00;
   ZEN2UV[3,36] := 16#00;
   ZEN2UV[3,37] := 16#00;
   ZEN2UV[3,38] := 16#00;
   ZEN2UV[3,39] := 16#00;
   ZEN2UV[3,40] := 16#00;
   ZEN2UV[3,41] := 16#00;
   ZEN2UV[3,42] := 16#00;
   ZEN2UV[3,43] := 16#00;
   ZEN2UV[3,44] := 16#00;
   ZEN2UV[3,45] := 16#00;
   ZEN2UV[3,46] := 16#00;
   ZEN2UV[3,47] := 16#00;
   ZEN2UV[3,48] := 16#00;
   ZEN2UV[3,49] := 16#00;
   ZEN2UV[3,50] := 16#00;
   ZEN2UV[3,51] := 16#00;
   ZEN2UV[3,52] := 16#00;
   ZEN2UV[3,53] := 16#00;
   ZEN2UV[3,54] := 16#00;
   ZEN2UV[3,55] := 16#00;
   ZEN2UV[3,56] := 16#00;
   ZEN2UV[3,57] := 16#00;
   ZEN2UV[3,58] := 16#00;
   ZEN2UV[3,59] := 16#00;
   ZEN2UV[3,60] := 16#00;
   ZEN2UV[3,61] := 16#00;
   ZEN2UV[3,62] := 16#00;
   ZEN2UV[3,63] := 16#00;
   ZEN2UV[3,64] := 16#00;
   ZEN2UV[3,65] := 16#00;
   ZEN2UV[3,66] := 16#00;
   ZEN2UV[3,67] := 16#00;
   ZEN2UV[3,68] := 16#00;
   ZEN2UV[3,69] := 16#00;
   ZEN2UV[3,70] := 16#00;
   ZEN2UV[3,71] := 16#00;
   ZEN2UV[3,72] := 16#00;
   ZEN2UV[3,73] := 16#00;
   ZEN2UV[3,74] := 16#00;
   ZEN2UV[3,75] := 16#00;
   ZEN2UV[3,76] := 16#00;
   ZEN2UV[3,77] := 16#00;
   ZEN2UV[3,78] := 16#00;
   ZEN2UV[3,79] := 16#00;
   ZEN2UV[3,80] := 16#00;
   ZEN2UV[3,81] := 16#00;
   ZEN2UV[3,82] := 16#00;
   ZEN2UV[3,83] := 16#00;
   ZEN2UV[3,84] := 16#00;
   ZEN2UV[3,85] := 16#00;
   ZEN2UV[3,86] := 16#00;
   ZEN2UV[3,87] := 16#00;
   ZEN2UV[3,88] := 16#00;
   ZEN2UV[3,89] := 16#00;
   ZEN2UV[3,90] := 16#00;
   ZEN2UV[3,91] := 16#00;
   ZEN2UV[3,92] := 16#00;
   ZEN2UV[3,93] := 16#00;
   ZEN2UV[3,94] := 16#00;
   ZEN2UV[3,95] := 16#00;
   ZEN2UV[3,96] := 16#00;
   ZEN2UV[3,97] := 16#00;
   ZEN2UV[3,98] := 16#00;
   ZEN2UV[3,99] := 16#00;
   ZEN2UV[3,100] := 16#00;
   ZEN2UV[3,101] := 16#00;
   ZEN2UV[3,102] := 16#00;
   ZEN2UV[3,103] := 16#00;
   ZEN2UV[3,104] := 16#00;
   ZEN2UV[3,105] := 16#00;
   ZEN2UV[3,106] := 16#00;
   ZEN2UV[3,107] := 16#00;
   ZEN2UV[3,108] := 16#00;
   ZEN2UV[3,109] := 16#00;
   ZEN2UV[3,110] := 16#00;
   ZEN2UV[3,111] := 16#00;
   ZEN2UV[3,112] := 16#00;
   ZEN2UV[3,113] := 16#00;
   ZEN2UV[3,114] := 16#00;
   ZEN2UV[3,115] := 16#00;
   ZEN2UV[3,116] := 16#00;
   ZEN2UV[3,117] := 16#00;
   ZEN2UV[3,118] := 16#00;
   ZEN2UV[3,119] := 16#00;
   ZEN2UV[3,120] := 16#00;
   ZEN2UV[3,121] := 16#00;
   ZEN2UV[3,122] := 16#00;
   ZEN2UV[3,123] := 16#00;
   ZEN2UV[3,124] := 16#00;
   ZEN2UV[3,125] := 16#00;
   ZEN2UV[3,126] := 16#00;
   ZEN2UV[3,127] := 16#00;
   ZEN2UV[3,128] := 16#00;
   ZEN2UV[3,129] := 16#00;
   ZEN2UV[3,130] := 16#00;
   ZEN2UV[3,131] := 16#00;
   ZEN2UV[3,132] := 16#00;
   ZEN2UV[4,1] := 16#00;
   ZEN2UV[4,2] := 16#00;
   ZEN2UV[4,3] := 16#00;
   ZEN2UV[4,4] := 16#00;
   ZEN2UV[4,5] := 16#00;
   ZEN2UV[4,6] := 16#00;
   ZEN2UV[4,7] := 16#00;
   ZEN2UV[4,8] := 16#00;
   ZEN2UV[4,9] := 16#00;
   ZEN2UV[4,10] := 16#00;
   ZEN2UV[4,11] := 16#00;
   ZEN2UV[4,12] := 16#00;
   ZEN2UV[4,13] := 16#00;
   ZEN2UV[4,14] := 16#00;
   ZEN2UV[4,15] := 16#00;
   ZEN2UV[4,16] := 16#00;
   ZEN2UV[4,17] := 16#00;
   ZEN2UV[4,18] := 16#00;
   ZEN2UV[4,19] := 16#00;
   ZEN2UV[4,20] := 16#00;
   ZEN2UV[4,21] := 16#00;
   ZEN2UV[4,22] := 16#00;
   ZEN2UV[4,23] := 16#00;
   ZEN2UV[4,24] := 16#00;
   ZEN2UV[4,25] := 16#00;
   ZEN2UV[4,26] := 16#00;
   ZEN2UV[4,27] := 16#00;
   ZEN2UV[4,28] := 16#00;
   ZEN2UV[4,29] := 16#00;
   ZEN2UV[4,30] := 16#00;
   ZEN2UV[4,31] := 16#00;
   ZEN2UV[4,32] := 16#00;
   ZEN2UV[4,33] := 16#00;
   ZEN2UV[4,34] := 16#00;
   ZEN2UV[4,35] := 16#00;
   ZEN2UV[4,36] := 16#00;
   ZEN2UV[4,37] := 16#00;
   ZEN2UV[4,38] := 16#00;
   ZEN2UV[4,39] := 16#00;
   ZEN2UV[4,40] := 16#00;
   ZEN2UV[4,41] := 16#00;
   ZEN2UV[4,42] := 16#00;
   ZEN2UV[4,43] := 16#00;
   ZEN2UV[4,44] := 16#00;
   ZEN2UV[4,45] := 16#00;
   ZEN2UV[4,46] := 16#00;
   ZEN2UV[4,47] := 16#00;
   ZEN2UV[4,48] := 16#00;
   ZEN2UV[4,49] := 16#00;
   ZEN2UV[4,50] := 16#00;
   ZEN2UV[4,51] := 16#00;
   ZEN2UV[4,52] := 16#00;
   ZEN2UV[4,53] := 16#00;
   ZEN2UV[4,54] := 16#00;
   ZEN2UV[4,55] := 16#00;
   ZEN2UV[4,56] := 16#00;
   ZEN2UV[4,57] := 16#00;
   ZEN2UV[4,58] := 16#00;
   ZEN2UV[4,59] := 16#00;
   ZEN2UV[4,60] := 16#00;
   ZEN2UV[4,61] := 16#00;
   ZEN2UV[4,62] := 16#00;
   ZEN2UV[4,63] := 16#00;
   ZEN2UV[4,64] := 16#00;
   ZEN2UV[4,65] := 16#00;
   ZEN2UV[4,66] := 16#00;
   ZEN2UV[4,67] := 16#00;
   ZEN2UV[4,68] := 16#00;
   ZEN2UV[4,69] := 16#00;
   ZEN2UV[4,70] := 16#00;
   ZEN2UV[4,71] := 16#00;
   ZEN2UV[4,72] := 16#00;
   ZEN2UV[4,73] := 16#00;
   ZEN2UV[4,74] := 16#00;
   ZEN2UV[4,75] := 16#00;
   ZEN2UV[4,76] := 16#00;
   ZEN2UV[4,77] := 16#00;
   ZEN2UV[4,78] := 16#00;
   ZEN2UV[4,79] := 16#00;
   ZEN2UV[4,80] := 16#00;
   ZEN2UV[4,81] := 16#00;
   ZEN2UV[4,82] := 16#00;
   ZEN2UV[4,83] := 16#00;
   ZEN2UV[4,84] := 16#00;
   ZEN2UV[4,85] := 16#00;
   ZEN2UV[4,86] := 16#00;
   ZEN2UV[4,87] := 16#00;
   ZEN2UV[4,88] := 16#00;
   ZEN2UV[4,89] := 16#00;
   ZEN2UV[4,90] := 16#00;
   ZEN2UV[4,91] := 16#00;
   ZEN2UV[4,92] := 16#00;
   ZEN2UV[4,93] := 16#00;
   ZEN2UV[4,94] := 16#00;
   ZEN2UV[4,95] := 16#00;
   ZEN2UV[4,96] := 16#00;
   ZEN2UV[4,97] := 16#00;
   ZEN2UV[4,98] := 16#00;
   ZEN2UV[4,99] := 16#00;
   ZEN2UV[4,100] := 16#00;
   ZEN2UV[4,101] := 16#00;
   ZEN2UV[4,102] := 16#00;
   ZEN2UV[4,103] := 16#00;
   ZEN2UV[4,104] := 16#00;
   ZEN2UV[4,105] := 16#00;
   ZEN2UV[4,106] := 16#00;
   ZEN2UV[4,107] := 16#00;
   ZEN2UV[4,108] := 16#00;
   ZEN2UV[4,109] := 16#00;
   ZEN2UV[4,110] := 16#00;
   ZEN2UV[4,111] := 16#00;
   ZEN2UV[4,112] := 16#00;
   ZEN2UV[4,113] := 16#00;
   ZEN2UV[4,114] := 16#00;
   ZEN2UV[4,115] := 16#00;
   ZEN2UV[4,116] := 16#00;
   ZEN2UV[4,117] := 16#00;
   ZEN2UV[4,118] := 16#00;
   ZEN2UV[4,119] := 16#00;
   ZEN2UV[4,120] := 16#00;
   ZEN2UV[4,121] := 16#00;
   ZEN2UV[4,122] := 16#00;
   ZEN2UV[4,123] := 16#00;
   ZEN2UV[4,124] := 16#00;
   ZEN2UV[4,125] := 16#00;
   ZEN2UV[4,126] := 16#00;
   ZEN2UV[4,127] := 16#00;
   ZEN2UV[4,128] := 16#00;
   ZEN2UV[4,129] := 16#00;
   ZEN2UV[4,130] := 16#00;
   ZEN2UV[4,131] := 16#00;
   ZEN2UV[4,132] := 16#00;
   ZEN2UV[5,1] := 16#00;
   ZEN2UV[5,2] := 16#00;
   ZEN2UV[5,3] := 16#00;
   ZEN2UV[5,4] := 16#00;
   ZEN2UV[5,5] := 16#00;
   ZEN2UV[5,6] := 16#00;
   ZEN2UV[5,7] := 16#00;
   ZEN2UV[5,8] := 16#00;
   ZEN2UV[5,9] := 16#00;
   ZEN2UV[5,10] := 16#00;
   ZEN2UV[5,11] := 16#00;
   ZEN2UV[5,12] := 16#00;
   ZEN2UV[5,13] := 16#00;
   ZEN2UV[5,14] := 16#00;
   ZEN2UV[5,15] := 16#00;
   ZEN2UV[5,16] := 16#00;
   ZEN2UV[5,17] := 16#00;
   ZEN2UV[5,18] := 16#00;
   ZEN2UV[5,19] := 16#00;
   ZEN2UV[5,20] := 16#00;
   ZEN2UV[5,21] := 16#00;
   ZEN2UV[5,22] := 16#00;
   ZEN2UV[5,23] := 16#00;
   ZEN2UV[5,24] := 16#00;
   ZEN2UV[5,25] := 16#00;
   ZEN2UV[5,26] := 16#00;
   ZEN2UV[5,27] := 16#00;
   ZEN2UV[5,28] := 16#00;
   ZEN2UV[5,29] := 16#00;
   ZEN2UV[5,30] := 16#00;
   ZEN2UV[5,31] := 16#00;
   ZEN2UV[5,32] := 16#00;
   ZEN2UV[5,33] := 16#00;
   ZEN2UV[5,34] := 16#00;
   ZEN2UV[5,35] := 16#00;
   ZEN2UV[5,36] := 16#00;
   ZEN2UV[5,37] := 16#00;
   ZEN2UV[5,38] := 16#00;
   ZEN2UV[5,39] := 16#00;
   ZEN2UV[5,40] := 16#00;
   ZEN2UV[5,41] := 16#00;
   ZEN2UV[5,42] := 16#00;
   ZEN2UV[5,43] := 16#00;
   ZEN2UV[5,44] := 16#00;
   ZEN2UV[5,45] := 16#00;
   ZEN2UV[5,46] := 16#00;
   ZEN2UV[5,47] := 16#00;
   ZEN2UV[5,48] := 16#00;
   ZEN2UV[5,49] := 16#00;
   ZEN2UV[5,50] := 16#00;
   ZEN2UV[5,51] := 16#00;
   ZEN2UV[5,52] := 16#00;
   ZEN2UV[5,53] := 16#00;
   ZEN2UV[5,54] := 16#00;
   ZEN2UV[5,55] := 16#00;
   ZEN2UV[5,56] := 16#00;
   ZEN2UV[5,57] := 16#00;
   ZEN2UV[5,58] := 16#00;
   ZEN2UV[5,59] := 16#00;
   ZEN2UV[5,60] := 16#00;
   ZEN2UV[5,61] := 16#00;
   ZEN2UV[5,62] := 16#00;
   ZEN2UV[5,63] := 16#00;
   ZEN2UV[5,64] := 16#00;
   ZEN2UV[5,65] := 16#00;
   ZEN2UV[5,66] := 16#00;
   ZEN2UV[5,67] := 16#00;
   ZEN2UV[5,68] := 16#00;
   ZEN2UV[5,69] := 16#00;
   ZEN2UV[5,70] := 16#00;
   ZEN2UV[5,71] := 16#00;
   ZEN2UV[5,72] := 16#00;
   ZEN2UV[5,73] := 16#00;
   ZEN2UV[5,74] := 16#00;
   ZEN2UV[5,75] := 16#00;
   ZEN2UV[5,76] := 16#00;
   ZEN2UV[5,77] := 16#00;
   ZEN2UV[5,78] := 16#00;
   ZEN2UV[5,79] := 16#00;
   ZEN2UV[5,80] := 16#00;
   ZEN2UV[5,81] := 16#00;
   ZEN2UV[5,82] := 16#00;
   ZEN2UV[5,83] := 16#00;
   ZEN2UV[5,84] := 16#00;
   ZEN2UV[5,85] := 16#00;
   ZEN2UV[5,86] := 16#00;
   ZEN2UV[5,87] := 16#00;
   ZEN2UV[5,88] := 16#00;
   ZEN2UV[5,89] := 16#00;
   ZEN2UV[5,90] := 16#00;
   ZEN2UV[5,91] := 16#00;
   ZEN2UV[5,92] := 16#00;
   ZEN2UV[5,93] := 16#00;
   ZEN2UV[5,94] := 16#00;
   ZEN2UV[5,95] := 16#00;
   ZEN2UV[5,96] := 16#00;
   ZEN2UV[5,97] := 16#00;
   ZEN2UV[5,98] := 16#00;
   ZEN2UV[5,99] := 16#00;
   ZEN2UV[5,100] := 16#00;
   ZEN2UV[5,101] := 16#00;
   ZEN2UV[5,102] := 16#00;
   ZEN2UV[5,103] := 16#00;
   ZEN2UV[5,104] := 16#00;
   ZEN2UV[5,105] := 16#00;
   ZEN2UV[5,106] := 16#00;
   ZEN2UV[5,107] := 16#00;
   ZEN2UV[5,108] := 16#00;
   ZEN2UV[5,109] := 16#00;
   ZEN2UV[5,110] := 16#00;
   ZEN2UV[5,111] := 16#00;
   ZEN2UV[5,112] := 16#00;
   ZEN2UV[5,113] := 16#00;
   ZEN2UV[5,114] := 16#00;
   ZEN2UV[5,115] := 16#00;
   ZEN2UV[5,116] := 16#00;
   ZEN2UV[5,117] := 16#00;
   ZEN2UV[5,118] := 16#00;
   ZEN2UV[5,119] := 16#00;
   ZEN2UV[5,120] := 16#00;
   ZEN2UV[5,121] := 16#00;
   ZEN2UV[5,122] := 16#00;
   ZEN2UV[5,123] := 16#00;
   ZEN2UV[5,124] := 16#00;
   ZEN2UV[5,125] := 16#00;
   ZEN2UV[5,126] := 16#00;
   ZEN2UV[5,127] := 16#00;
   ZEN2UV[5,128] := 16#00;
   ZEN2UV[5,129] := 16#00;
   ZEN2UV[5,130] := 16#00;
   ZEN2UV[5,131] := 16#00;
   ZEN2UV[5,132] := 16#00;
   ZEN2UV[6,1] := 16#00;
   ZEN2UV[6,2] := 16#00;
   ZEN2UV[6,3] := 16#00;
   ZEN2UV[6,4] := 16#00;
   ZEN2UV[6,5] := 16#00;
   ZEN2UV[6,6] := 16#00;
   ZEN2UV[6,7] := 16#00;
   ZEN2UV[6,8] := 16#00;
   ZEN2UV[6,9] := 16#00;
   ZEN2UV[6,10] := 16#00;
   ZEN2UV[6,11] := 16#00;
   ZEN2UV[6,12] := 16#00;
   ZEN2UV[6,13] := 16#00;
   ZEN2UV[6,14] := 16#00;
   ZEN2UV[6,15] := 16#00;
   ZEN2UV[6,16] := 16#00;
   ZEN2UV[6,17] := 16#00;
   ZEN2UV[6,18] := 16#00;
   ZEN2UV[6,19] := 16#00;
   ZEN2UV[6,20] := 16#00;
   ZEN2UV[6,21] := 16#00;
   ZEN2UV[6,22] := 16#00;
   ZEN2UV[6,23] := 16#00;
   ZEN2UV[6,24] := 16#00;
   ZEN2UV[6,25] := 16#00;
   ZEN2UV[6,26] := 16#00;
   ZEN2UV[6,27] := 16#00;
   ZEN2UV[6,28] := 16#00;
   ZEN2UV[6,29] := 16#00;
   ZEN2UV[6,30] := 16#00;
   ZEN2UV[6,31] := 16#00;
   ZEN2UV[6,32] := 16#00;
   ZEN2UV[6,33] := 16#00;
   ZEN2UV[6,34] := 16#00;
   ZEN2UV[6,35] := 16#00;
   ZEN2UV[6,36] := 16#00;
   ZEN2UV[6,37] := 16#00;
   ZEN2UV[6,38] := 16#00;
   ZEN2UV[6,39] := 16#00;
   ZEN2UV[6,40] := 16#00;
   ZEN2UV[6,41] := 16#01;
   ZEN2UV[6,42] := 16#02;
   ZEN2UV[6,43] := 16#03;
   ZEN2UV[6,44] := 16#00;
   ZEN2UV[6,45] := 16#00;
   ZEN2UV[6,46] := 16#00;
   ZEN2UV[6,47] := 16#00;
   ZEN2UV[6,48] := 16#00;
   ZEN2UV[6,49] := 16#00;
   ZEN2UV[6,50] := 16#00;
   ZEN2UV[6,51] := 16#00;
   ZEN2UV[6,52] := 16#00;
   ZEN2UV[6,53] := 16#00;
   ZEN2UV[6,54] := 16#00;
   ZEN2UV[6,55] := 16#00;
   ZEN2UV[6,56] := 16#00;
   ZEN2UV[6,57] := 16#00;
   ZEN2UV[6,58] := 16#00;
   ZEN2UV[6,59] := 16#00;
   ZEN2UV[6,60] := 16#00;
   ZEN2UV[6,61] := 16#00;
   ZEN2UV[6,62] := 16#00;
   ZEN2UV[6,63] := 16#04;
   ZEN2UV[6,64] := 16#05;
   ZEN2UV[6,65] := 16#06;
   ZEN2UV[6,66] := 16#07;
   ZEN2UV[6,67] := 16#08;
   ZEN2UV[6,68] := 16#09;
   ZEN2UV[6,69] := 16#0A;
   ZEN2UV[6,70] := 16#0B;
   ZEN2UV[6,71] := 16#0C;
   ZEN2UV[6,72] := 16#0D;
   ZEN2UV[6,73] := 16#0E;
   ZEN2UV[6,74] := 16#0F;
   ZEN2UV[6,75] := 16#10;
   ZEN2UV[6,76] := 16#11;
   ZEN2UV[6,77] := 16#12;
   ZEN2UV[6,78] := 16#13;
   ZEN2UV[6,79] := 16#14;
   ZEN2UV[6,80] := 16#15;
   ZEN2UV[6,81] := 16#16;
   ZEN2UV[6,82] := 16#17;
   ZEN2UV[6,83] := 16#18;
   ZEN2UV[6,84] := 16#19;
   ZEN2UV[6,85] := 16#1A;
   ZEN2UV[6,86] := 16#1B;
   ZEN2UV[6,87] := 16#1C;
   ZEN2UV[6,88] := 16#1D;
   ZEN2UV[6,89] := 16#1E;
   ZEN2UV[6,90] := 16#1F;
   ZEN2UV[6,91] := 16#20;
   ZEN2UV[6,92] := 16#21;
   ZEN2UV[6,93] := 16#22;
   ZEN2UV[6,94] := 16#23;
   ZEN2UV[6,95] := 16#24;
   ZEN2UV[6,96] := 16#25;
   ZEN2UV[6,97] := 16#26;
   ZEN2UV[6,98] := 16#00;
   ZEN2UV[6,99] := 16#00;
   ZEN2UV[6,100] := 16#00;
   ZEN2UV[6,101] := 16#00;
   ZEN2UV[6,102] := 16#00;
   ZEN2UV[6,103] := 16#00;
   ZEN2UV[6,104] := 16#00;
   ZEN2UV[6,105] := 16#00;
   ZEN2UV[6,106] := 16#00;
   ZEN2UV[6,107] := 16#00;
   ZEN2UV[6,108] := 16#00;
   ZEN2UV[6,109] := 16#00;
   ZEN2UV[6,110] := 16#00;
   ZEN2UV[6,111] := 16#00;
   ZEN2UV[6,112] := 16#00;
   ZEN2UV[6,113] := 16#00;
   ZEN2UV[6,114] := 16#00;
   ZEN2UV[6,115] := 16#00;
   ZEN2UV[6,116] := 16#00;
   ZEN2UV[6,117] := 16#00;
   ZEN2UV[6,118] := 16#00;
   ZEN2UV[6,119] := 16#00;
   ZEN2UV[6,120] := 16#00;
   ZEN2UV[6,121] := 16#00;
   ZEN2UV[6,122] := 16#00;
   ZEN2UV[6,123] := 16#00;
   ZEN2UV[6,124] := 16#00;
   ZEN2UV[6,125] := 16#00;
   ZEN2UV[6,126] := 16#00;
   ZEN2UV[6,127] := 16#00;
   ZEN2UV[6,128] := 16#00;
   ZEN2UV[6,129] := 16#00;
   ZEN2UV[6,130] := 16#00;
   ZEN2UV[6,131] := 16#00;
   ZEN2UV[6,132] := 16#00;

END_DATA_BLOCK

DATA_BLOCK "DB_IEC_Para_MAo_SP"
{ S7_Optimized_Access := 'FALSE' }
AUTHOR : SIE_GST
FAMILY : S7_IEC
NAME : P_NA_IM
VERSION : 1.6
   STRUCT
      DB_Manag { ExternalVisible := 'False'} : Struct
         Pos_of_DB { ExternalVisible := 'False'} : Byte;   // reserved for future - do not change !
         No_of_all_DBs { ExternalVisible := 'False'} : Byte;   // reserved for future - do not change !
         DB_No_Act { ExternalVisible := 'False'} : Word;   // reserved for future - do not change !
         DB_No_Prev { ExternalVisible := 'False'} : Word;   // reserved for future - do not change !
         DB_No_Next { ExternalVisible := 'False'} : Word;   // reserved for future - do not change !
         Reserved { ExternalVisible := 'False'} : Word;
      END_STRUCT;
      Info_Manag { ExternalVisible := 'False'} : Struct
         P_Byte_First_Info { ExternalVisible := 'False'} : Int;   // (Byte-) Position of first Para-Block - do not change !
         No_of_Infos { ExternalVisible := 'False'} : Int;   // 0:unspecified (DB is filled up to the end); otherwise size n of ARRAY [1..n]
         Len_Info { ExternalVisible := 'False'} : USInt;   // Difference in [byte] between two Para-Blocks - do not change !
         Len_Sort_Key { ExternalVisible := 'False'} : USInt;   // 0: without sorting; >0: Data sets are sorted ascending with x bytes
         Re_internal_usage { ExternalVisible := 'False'} : DWord;
      END_STRUCT;
      Global { ExternalVisible := 'False'} : Struct
         Para_DB_Type { ExternalVisible := 'False'} : Word;   // Internal identifier for this Data Block - do not change
         Image_Type { ExternalVisible := 'False'} : Byte;   // 1 Bit-Image, 2 IEC-Image, 3 IEC+Ext_State+Time
         Image_Len { ExternalVisible := 'False'} : Byte;   // 0: auto (standard); <> 0: fixed distance [Bit] of procesimages
         Subst_on_Error { ExternalVisible := 'False'} : Bool;   // Substitute values in case of connection errors ?
         Subst_Value { ExternalVisible := 'False'} : DWord;   // Substitute value (if activated). For SP only 0 and 1 possible
         Internal_10 { ExternalVisible := 'False'} : Word;   // Internal use: Last found parablock - do not change !
         Internal_12 { ExternalVisible := 'False'} : Word;   // Internal use: Last processed info - do not change !
      END_STRUCT;
      Para { ExternalVisible := 'False'} : Array[1..150] of Struct
         S_Line { ExternalVisible := 'False'} : Int;   // Source (Quelle): No of Line (Nr der Linie) (1..x)-actually do not change from 1
         S_ASDU { ExternalVisible := 'False'} : UInt;   // Source (Quelle): Address of ASDU (ASDU-Adresse)
         S_Info { ExternalVisible := 'False'} : DInt;   // Source (Quelle): Address of Infoobject (IOA)
         D_DB_No { ExternalVisible := 'False'} : Int;   // Dest. (Ziel) No. of DataBlock, 0 -> PIQ (PAA)
         D_Address { ExternalVisible := 'False'} : DInt;   // Dest. (Ziel): Bitposition
         P_No_of_fol_Infos { ExternalVisible := 'False'} : Int;   // Parameter: Number of following sequ. Infoelements
      END_STRUCT;
   END_STRUCT;


BEGIN
   Info_Manag.P_Byte_First_Info := 34;
   Info_Manag.No_of_Infos := 150;
   Info_Manag.Len_Info := 16;
   Global.Para_DB_Type := WORD#16#0101;
   Global.Image_Type := BYTE#16#03;
   Para[1].S_Line := 1;
   Para[1].S_ASDU := 25860;
   Para[1].S_Info := 240;
   Para[1].D_DB_No := 402;
   Para[2].S_Line := 1;
   Para[2].S_ASDU := 25860;
   Para[2].S_Info := 241;
   Para[2].D_DB_No := 402;
   Para[2].D_Address := 80;
   Para[3].S_Line := 1;
   Para[3].S_ASDU := 25860;
   Para[3].S_Info := 242;
   Para[3].D_DB_No := 402;
   Para[3].D_Address := 160;
   Para[4].S_Line := 1;
   Para[4].S_ASDU := 25860;
   Para[4].S_Info := 243;
   Para[4].D_DB_No := 402;
   Para[4].D_Address := 240;
   Para[5].S_Line := 1;
   Para[5].S_ASDU := 25860;
   Para[5].S_Info := 2;
   Para[5].D_DB_No := 402;
   Para[5].D_Address := 320;
   Para[6].S_Line := 1;
   Para[6].S_ASDU := 25860;
   Para[6].S_Info := 3;
   Para[6].D_DB_No := 402;
   Para[6].D_Address := 400;
   Para[7].S_Line := 1;
   Para[7].S_ASDU := 25860;
   Para[7].S_Info := 4;
   Para[7].D_DB_No := 402;
   Para[7].D_Address := 480;
   Para[8].S_Line := 1;
   Para[8].S_ASDU := 25860;
   Para[8].S_Info := 5;
   Para[8].D_DB_No := 402;
   Para[8].D_Address := 560;
   Para[9].S_Line := 1;
   Para[9].S_ASDU := 25860;
   Para[9].S_Info := 6;
   Para[9].D_DB_No := 402;
   Para[9].D_Address := 640;
   Para[10].S_Line := 1;
   Para[10].S_ASDU := 25860;
   Para[10].S_Info := 7;
   Para[10].D_DB_No := 402;
   Para[10].D_Address := 720;
   Para[11].S_Line := 1;
   Para[11].S_ASDU := 26116;
   Para[11].S_Info := 240;
   Para[11].D_DB_No := 402;
   Para[11].D_Address := 1216;
   Para[12].S_Line := 1;
   Para[12].S_ASDU := 26116;
   Para[12].S_Info := 241;
   Para[12].D_DB_No := 402;
   Para[12].D_Address := 1296;
   Para[13].S_Line := 1;
   Para[13].S_ASDU := 26116;
   Para[13].S_Info := 242;
   Para[13].D_DB_No := 402;
   Para[13].D_Address := 1376;
   Para[14].S_Line := 1;
   Para[14].S_ASDU := 26116;
   Para[14].S_Info := 243;
   Para[14].D_DB_No := 402;
   Para[14].D_Address := 1456;
   Para[15].S_Line := 1;
   Para[15].S_ASDU := 26116;
   Para[15].S_Info := 2;
   Para[15].D_DB_No := 402;
   Para[15].D_Address := 1536;
   Para[16].S_Line := 1;
   Para[16].S_ASDU := 26116;
   Para[16].S_Info := 3;
   Para[16].D_DB_No := 402;
   Para[16].D_Address := 1616;
   Para[17].S_Line := 1;
   Para[17].S_ASDU := 26116;
   Para[17].S_Info := 4;
   Para[17].D_DB_No := 402;
   Para[17].D_Address := 1696;
   Para[18].S_Line := 1;
   Para[18].S_ASDU := 26116;
   Para[18].S_Info := 5;
   Para[18].D_DB_No := 402;
   Para[18].D_Address := 1776;
   Para[19].S_Line := 1;
   Para[19].S_ASDU := 26116;
   Para[19].S_Info := 6;
   Para[19].D_DB_No := 402;
   Para[19].D_Address := 1856;
   Para[20].S_Line := 1;
   Para[20].S_ASDU := 26116;
   Para[20].S_Info := 7;
   Para[20].D_DB_No := 402;
   Para[20].D_Address := 1936;
   Para[21].S_Line := 1;
   Para[21].S_ASDU := 26372;
   Para[21].S_Info := 240;
   Para[21].D_DB_No := 402;
   Para[21].D_Address := 2432;
   Para[22].S_Line := 1;
   Para[22].S_ASDU := 26372;
   Para[22].S_Info := 241;
   Para[22].D_DB_No := 402;
   Para[22].D_Address := 2512;
   Para[23].S_Line := 1;
   Para[23].S_ASDU := 26372;
   Para[23].S_Info := 242;
   Para[23].D_DB_No := 402;
   Para[23].D_Address := 2592;
   Para[24].S_Line := 1;
   Para[24].S_ASDU := 26372;
   Para[24].S_Info := 243;
   Para[24].D_DB_No := 402;
   Para[24].D_Address := 2672;
   Para[25].S_Line := 1;
   Para[25].S_ASDU := 26372;
   Para[25].S_Info := 2;
   Para[25].D_DB_No := 402;
   Para[25].D_Address := 2752;
   Para[26].S_Line := 1;
   Para[26].S_ASDU := 26372;
   Para[26].S_Info := 3;
   Para[26].D_DB_No := 402;
   Para[26].D_Address := 2832;
   Para[27].S_Line := 1;
   Para[27].S_ASDU := 26372;
   Para[27].S_Info := 4;
   Para[27].D_DB_No := 402;
   Para[27].D_Address := 2912;
   Para[28].S_Line := 1;
   Para[28].S_ASDU := 26372;
   Para[28].S_Info := 5;
   Para[28].D_DB_No := 402;
   Para[28].D_Address := 2992;
   Para[29].S_Line := 1;
   Para[29].S_ASDU := 26372;
   Para[29].S_Info := 6;
   Para[29].D_DB_No := 402;
   Para[29].D_Address := 3072;
   Para[30].S_Line := 1;
   Para[30].S_ASDU := 26372;
   Para[30].S_Info := 7;
   Para[30].D_DB_No := 402;
   Para[30].D_Address := 3152;
   Para[31].S_Line := 1;
   Para[31].S_ASDU := 26628;
   Para[31].S_Info := 240;
   Para[31].D_DB_No := 402;
   Para[31].D_Address := 3648;
   Para[32].S_Line := 1;
   Para[32].S_ASDU := 26628;
   Para[32].S_Info := 241;
   Para[32].D_DB_No := 402;
   Para[32].D_Address := 3728;
   Para[33].S_Line := 1;
   Para[33].S_ASDU := 26628;
   Para[33].S_Info := 242;
   Para[33].D_DB_No := 402;
   Para[33].D_Address := 3808;
   Para[34].S_Line := 1;
   Para[34].S_ASDU := 26628;
   Para[34].S_Info := 243;
   Para[34].D_DB_No := 402;
   Para[34].D_Address := 3888;
   Para[35].S_Line := 1;
   Para[35].S_ASDU := 26628;
   Para[35].S_Info := 2;
   Para[35].D_DB_No := 402;
   Para[35].D_Address := 3968;
   Para[36].S_Line := 1;
   Para[36].S_ASDU := 26628;
   Para[36].S_Info := 3;
   Para[36].D_DB_No := 402;
   Para[36].D_Address := 4048;
   Para[37].S_Line := 1;
   Para[37].S_ASDU := 26628;
   Para[37].S_Info := 4;
   Para[37].D_DB_No := 402;
   Para[37].D_Address := 4128;
   Para[38].S_Line := 1;
   Para[38].S_ASDU := 26628;
   Para[38].S_Info := 5;
   Para[38].D_DB_No := 402;
   Para[38].D_Address := 4208;
   Para[39].S_Line := 1;
   Para[39].S_ASDU := 26628;
   Para[39].S_Info := 6;
   Para[39].D_DB_No := 402;
   Para[39].D_Address := 4288;
   Para[40].S_Line := 1;
   Para[40].S_ASDU := 26628;
   Para[40].S_Info := 7;
   Para[40].D_DB_No := 402;
   Para[40].D_Address := 4368;
   Para[41].S_Line := 1;
   Para[41].S_ASDU := 26884;
   Para[41].S_Info := 240;
   Para[41].D_DB_No := 402;
   Para[41].D_Address := 4864;
   Para[42].S_Line := 1;
   Para[42].S_ASDU := 26884;
   Para[42].S_Info := 241;
   Para[42].D_DB_No := 402;
   Para[42].D_Address := 4944;
   Para[43].S_Line := 1;
   Para[43].S_ASDU := 26884;
   Para[43].S_Info := 242;
   Para[43].D_DB_No := 402;
   Para[43].D_Address := 5024;
   Para[44].S_Line := 1;
   Para[44].S_ASDU := 26884;
   Para[44].S_Info := 243;
   Para[44].D_DB_No := 402;
   Para[44].D_Address := 5104;
   Para[45].S_Line := 1;
   Para[45].S_ASDU := 26884;
   Para[45].S_Info := 2;
   Para[45].D_DB_No := 402;
   Para[45].D_Address := 5184;
   Para[46].S_Line := 1;
   Para[46].S_ASDU := 26884;
   Para[46].S_Info := 3;
   Para[46].D_DB_No := 402;
   Para[46].D_Address := 5264;
   Para[47].S_Line := 1;
   Para[47].S_ASDU := 26884;
   Para[47].S_Info := 4;
   Para[47].D_DB_No := 402;
   Para[47].D_Address := 5344;
   Para[48].S_Line := 1;
   Para[48].S_ASDU := 26884;
   Para[48].S_Info := 5;
   Para[48].D_DB_No := 402;
   Para[48].D_Address := 5424;
   Para[49].S_Line := 1;
   Para[49].S_ASDU := 26884;
   Para[49].S_Info := 6;
   Para[49].D_DB_No := 402;
   Para[49].D_Address := 5504;
   Para[50].S_Line := 1;
   Para[50].S_ASDU := 26884;
   Para[50].S_Info := 7;
   Para[50].D_DB_No := 402;
   Para[50].D_Address := 5584;
   Para[51].S_Line := 1;
   Para[51].S_ASDU := 27140;
   Para[51].S_Info := 240;
   Para[51].D_DB_No := 402;
   Para[51].D_Address := 6080;
   Para[52].S_Line := 1;
   Para[52].S_ASDU := 27140;
   Para[52].S_Info := 241;
   Para[52].D_DB_No := 402;
   Para[52].D_Address := 6160;
   Para[53].S_Line := 1;
   Para[53].S_ASDU := 27140;
   Para[53].S_Info := 242;
   Para[53].D_DB_No := 402;
   Para[53].D_Address := 6240;
   Para[54].S_Line := 1;
   Para[54].S_ASDU := 27140;
   Para[54].S_Info := 243;
   Para[54].D_DB_No := 402;
   Para[54].D_Address := 6320;
   Para[55].S_Line := 1;
   Para[55].S_ASDU := 27140;
   Para[55].S_Info := 2;
   Para[55].D_DB_No := 402;
   Para[55].D_Address := 6400;
   Para[56].S_Line := 1;
   Para[56].S_ASDU := 27140;
   Para[56].S_Info := 3;
   Para[56].D_DB_No := 402;
   Para[56].D_Address := 6480;
   Para[57].S_Line := 1;
   Para[57].S_ASDU := 27140;
   Para[57].S_Info := 4;
   Para[57].D_DB_No := 402;
   Para[57].D_Address := 6560;
   Para[58].S_Line := 1;
   Para[58].S_ASDU := 27140;
   Para[58].S_Info := 5;
   Para[58].D_DB_No := 402;
   Para[58].D_Address := 6640;
   Para[59].S_Line := 1;
   Para[59].S_ASDU := 27140;
   Para[59].S_Info := 6;
   Para[59].D_DB_No := 402;
   Para[59].D_Address := 6720;
   Para[60].S_Line := 1;
   Para[60].S_ASDU := 27140;
   Para[60].S_Info := 7;
   Para[60].D_DB_No := 402;
   Para[60].D_Address := 6800;
   Para[61].S_Line := 1;
   Para[61].S_ASDU := 27396;
   Para[61].S_Info := 240;
   Para[61].D_DB_No := 402;
   Para[61].D_Address := 7296;
   Para[62].S_Line := 1;
   Para[62].S_ASDU := 27396;
   Para[62].S_Info := 241;
   Para[62].D_DB_No := 402;
   Para[62].D_Address := 7376;
   Para[63].S_Line := 1;
   Para[63].S_ASDU := 27396;
   Para[63].S_Info := 242;
   Para[63].D_DB_No := 402;
   Para[63].D_Address := 7456;
   Para[64].S_Line := 1;
   Para[64].S_ASDU := 27396;
   Para[64].S_Info := 243;
   Para[64].D_DB_No := 402;
   Para[64].D_Address := 7536;
   Para[65].S_Line := 1;
   Para[65].S_ASDU := 27396;
   Para[65].S_Info := 2;
   Para[65].D_DB_No := 402;
   Para[65].D_Address := 7616;
   Para[66].S_Line := 1;
   Para[66].S_ASDU := 27396;
   Para[66].S_Info := 3;
   Para[66].D_DB_No := 402;
   Para[66].D_Address := 7696;
   Para[67].S_Line := 1;
   Para[67].S_ASDU := 27396;
   Para[67].S_Info := 4;
   Para[67].D_DB_No := 402;
   Para[67].D_Address := 7776;
   Para[68].S_Line := 1;
   Para[68].S_ASDU := 27396;
   Para[68].S_Info := 5;
   Para[68].D_DB_No := 402;
   Para[68].D_Address := 7856;
   Para[69].S_Line := 1;
   Para[69].S_ASDU := 27396;
   Para[69].S_Info := 6;
   Para[69].D_DB_No := 402;
   Para[69].D_Address := 7936;
   Para[70].S_Line := 1;
   Para[70].S_ASDU := 27396;
   Para[70].S_Info := 7;
   Para[70].D_DB_No := 402;
   Para[70].D_Address := 8016;
   Para[71].S_Line := 1;
   Para[71].S_ASDU := 27652;
   Para[71].S_Info := 240;
   Para[71].D_DB_No := 402;
   Para[71].D_Address := 8512;
   Para[72].S_Line := 1;
   Para[72].S_ASDU := 27652;
   Para[72].S_Info := 241;
   Para[72].D_DB_No := 402;
   Para[72].D_Address := 8592;
   Para[73].S_Line := 1;
   Para[73].S_ASDU := 27652;
   Para[73].S_Info := 242;
   Para[73].D_DB_No := 402;
   Para[73].D_Address := 8672;
   Para[74].S_Line := 1;
   Para[74].S_ASDU := 27652;
   Para[74].S_Info := 243;
   Para[74].D_DB_No := 402;
   Para[74].D_Address := 8752;
   Para[75].S_Line := 1;
   Para[75].S_ASDU := 27652;
   Para[75].S_Info := 2;
   Para[75].D_DB_No := 402;
   Para[75].D_Address := 8832;
   Para[76].S_Line := 1;
   Para[76].S_ASDU := 27652;
   Para[76].S_Info := 3;
   Para[76].D_DB_No := 402;
   Para[76].D_Address := 8912;
   Para[77].S_Line := 1;
   Para[77].S_ASDU := 27652;
   Para[77].S_Info := 4;
   Para[77].D_DB_No := 402;
   Para[77].D_Address := 8992;
   Para[78].S_Line := 1;
   Para[78].S_ASDU := 27652;
   Para[78].S_Info := 5;
   Para[78].D_DB_No := 402;
   Para[78].D_Address := 9072;
   Para[79].S_Line := 1;
   Para[79].S_ASDU := 27652;
   Para[79].S_Info := 6;
   Para[79].D_DB_No := 402;
   Para[79].D_Address := 9152;
   Para[80].S_Line := 1;
   Para[80].S_ASDU := 27652;
   Para[80].S_Info := 7;
   Para[80].D_DB_No := 402;
   Para[80].D_Address := 9232;
   Para[81].S_Line := 1;
   Para[81].S_ASDU := 28164;
   Para[81].S_Info := 240;
   Para[81].D_DB_No := 402;
   Para[81].D_Address := 9728;
   Para[82].S_Line := 1;
   Para[82].S_ASDU := 28164;
   Para[82].S_Info := 241;
   Para[82].D_DB_No := 402;
   Para[82].D_Address := 9808;
   Para[83].S_Line := 1;
   Para[83].S_ASDU := 28164;
   Para[83].S_Info := 242;
   Para[83].D_DB_No := 402;
   Para[83].D_Address := 9888;
   Para[84].S_Line := 1;
   Para[84].S_ASDU := 28164;
   Para[84].S_Info := 243;
   Para[84].D_DB_No := 402;
   Para[84].D_Address := 9968;
   Para[85].S_Line := 1;
   Para[85].S_ASDU := 28164;
   Para[85].S_Info := 2;
   Para[85].D_DB_No := 402;
   Para[85].D_Address := 10048;
   Para[86].S_Line := 1;
   Para[86].S_ASDU := 28164;
   Para[86].S_Info := 3;
   Para[86].D_DB_No := 402;
   Para[86].D_Address := 10128;
   Para[87].S_Line := 1;
   Para[87].S_ASDU := 28164;
   Para[87].S_Info := 4;
   Para[87].D_DB_No := 402;
   Para[87].D_Address := 10208;
   Para[88].S_Line := 1;
   Para[88].S_ASDU := 28164;
   Para[88].S_Info := 5;
   Para[88].D_DB_No := 402;
   Para[88].D_Address := 10288;
   Para[89].S_Line := 1;
   Para[89].S_ASDU := 28164;
   Para[89].S_Info := 6;
   Para[89].D_DB_No := 402;
   Para[89].D_Address := 10368;
   Para[90].S_Line := 1;
   Para[90].S_ASDU := 28164;
   Para[90].S_Info := 7;
   Para[90].D_DB_No := 402;
   Para[90].D_Address := 10448;
   Para[91].S_Line := 1;
   Para[91].S_ASDU := 28420;
   Para[91].S_Info := 240;
   Para[91].D_DB_No := 402;
   Para[91].D_Address := 10944;
   Para[92].S_Line := 1;
   Para[92].S_ASDU := 28420;
   Para[92].S_Info := 241;
   Para[92].D_DB_No := 402;
   Para[92].D_Address := 11024;
   Para[93].S_Line := 1;
   Para[93].S_ASDU := 28420;
   Para[93].S_Info := 242;
   Para[93].D_DB_No := 402;
   Para[93].D_Address := 11104;
   Para[94].S_Line := 1;
   Para[94].S_ASDU := 28420;
   Para[94].S_Info := 243;
   Para[94].D_DB_No := 402;
   Para[94].D_Address := 11184;
   Para[95].S_Line := 1;
   Para[95].S_ASDU := 28420;
   Para[95].S_Info := 2;
   Para[95].D_DB_No := 402;
   Para[95].D_Address := 11264;
   Para[96].S_Line := 1;
   Para[96].S_ASDU := 28420;
   Para[96].S_Info := 3;
   Para[96].D_DB_No := 402;
   Para[96].D_Address := 11344;
   Para[97].S_Line := 1;
   Para[97].S_ASDU := 28420;
   Para[97].S_Info := 4;
   Para[97].D_DB_No := 402;
   Para[97].D_Address := 11424;
   Para[98].S_Line := 1;
   Para[98].S_ASDU := 28420;
   Para[98].S_Info := 5;
   Para[98].D_DB_No := 402;
   Para[98].D_Address := 11504;
   Para[99].S_Line := 1;
   Para[99].S_ASDU := 28420;
   Para[99].S_Info := 6;
   Para[99].D_DB_No := 402;
   Para[99].D_Address := 11584;
   Para[100].S_Line := 1;
   Para[100].S_ASDU := 28420;
   Para[100].S_Info := 7;
   Para[100].D_DB_No := 402;
   Para[100].D_Address := 11664;
   Para[101].S_Line := 1;
   Para[101].S_ASDU := 28676;
   Para[101].S_Info := 240;
   Para[101].D_DB_No := 402;
   Para[101].D_Address := 12160;
   Para[102].S_Line := 1;
   Para[102].S_ASDU := 28676;
   Para[102].S_Info := 241;
   Para[102].D_DB_No := 402;
   Para[102].D_Address := 12240;
   Para[103].S_Line := 1;
   Para[103].S_ASDU := 28676;
   Para[103].S_Info := 242;
   Para[103].D_DB_No := 402;
   Para[103].D_Address := 12320;
   Para[104].S_Line := 1;
   Para[104].S_ASDU := 28676;
   Para[104].S_Info := 243;
   Para[104].D_DB_No := 402;
   Para[104].D_Address := 12400;
   Para[105].S_Line := 1;
   Para[105].S_ASDU := 28676;
   Para[105].S_Info := 2;
   Para[105].D_DB_No := 402;
   Para[105].D_Address := 12480;
   Para[106].S_Line := 1;
   Para[106].S_ASDU := 28676;
   Para[106].S_Info := 3;
   Para[106].D_DB_No := 402;
   Para[106].D_Address := 12560;
   Para[107].S_Line := 1;
   Para[107].S_ASDU := 28676;
   Para[107].S_Info := 4;
   Para[107].D_DB_No := 402;
   Para[107].D_Address := 12640;
   Para[108].S_Line := 1;
   Para[108].S_ASDU := 28676;
   Para[108].S_Info := 5;
   Para[108].D_DB_No := 402;
   Para[108].D_Address := 12720;
   Para[109].S_Line := 1;
   Para[109].S_ASDU := 28676;
   Para[109].S_Info := 6;
   Para[109].D_DB_No := 402;
   Para[109].D_Address := 12800;
   Para[110].S_Line := 1;
   Para[110].S_ASDU := 28676;
   Para[110].S_Info := 7;
   Para[110].D_DB_No := 402;
   Para[110].D_Address := 12880;
   Para[111].S_Line := 1;
   Para[111].S_ASDU := 28932;
   Para[111].S_Info := 240;
   Para[111].D_DB_No := 402;
   Para[111].D_Address := 13376;
   Para[112].S_Line := 1;
   Para[112].S_ASDU := 28932;
   Para[112].S_Info := 241;
   Para[112].D_DB_No := 402;
   Para[112].D_Address := 13456;
   Para[113].S_Line := 1;
   Para[113].S_ASDU := 28932;
   Para[113].S_Info := 242;
   Para[113].D_DB_No := 402;
   Para[113].D_Address := 13536;
   Para[114].S_Line := 1;
   Para[114].S_ASDU := 28932;
   Para[114].S_Info := 243;
   Para[114].D_DB_No := 402;
   Para[114].D_Address := 13616;
   Para[115].S_Line := 1;
   Para[115].S_ASDU := 28932;
   Para[115].S_Info := 2;
   Para[115].D_DB_No := 402;
   Para[115].D_Address := 13696;
   Para[116].S_Line := 1;
   Para[116].S_ASDU := 28932;
   Para[116].S_Info := 3;
   Para[116].D_DB_No := 402;
   Para[116].D_Address := 13776;
   Para[117].S_Line := 1;
   Para[117].S_ASDU := 28932;
   Para[117].S_Info := 4;
   Para[117].D_DB_No := 402;
   Para[117].D_Address := 13856;
   Para[118].S_Line := 1;
   Para[118].S_ASDU := 28932;
   Para[118].S_Info := 5;
   Para[118].D_DB_No := 402;
   Para[118].D_Address := 13936;
   Para[119].S_Line := 1;
   Para[119].S_ASDU := 28932;
   Para[119].S_Info := 6;
   Para[119].D_DB_No := 402;
   Para[119].D_Address := 14016;
   Para[120].S_Line := 1;
   Para[120].S_ASDU := 28932;
   Para[120].S_Info := 7;
   Para[120].D_DB_No := 402;
   Para[120].D_Address := 14096;
   Para[121].S_Line := 1;
   Para[121].S_ASDU := 29188;
   Para[121].S_Info := 240;
   Para[121].D_DB_No := 402;
   Para[121].D_Address := 14592;
   Para[122].S_Line := 1;
   Para[122].S_ASDU := 29188;
   Para[122].S_Info := 241;
   Para[122].D_DB_No := 402;
   Para[122].D_Address := 14672;
   Para[123].S_Line := 1;
   Para[123].S_ASDU := 29188;
   Para[123].S_Info := 242;
   Para[123].D_DB_No := 402;
   Para[123].D_Address := 14752;
   Para[124].S_Line := 1;
   Para[124].S_ASDU := 29188;
   Para[124].S_Info := 243;
   Para[124].D_DB_No := 402;
   Para[124].D_Address := 14832;
   Para[125].S_Line := 1;
   Para[125].S_ASDU := 29188;
   Para[125].S_Info := 2;
   Para[125].D_DB_No := 402;
   Para[125].D_Address := 14912;
   Para[126].S_Line := 1;
   Para[126].S_ASDU := 29188;
   Para[126].S_Info := 3;
   Para[126].D_DB_No := 402;
   Para[126].D_Address := 14992;
   Para[127].S_Line := 1;
   Para[127].S_ASDU := 29188;
   Para[127].S_Info := 4;
   Para[127].D_DB_No := 402;
   Para[127].D_Address := 15072;
   Para[128].S_Line := 1;
   Para[128].S_ASDU := 29188;
   Para[128].S_Info := 5;
   Para[128].D_DB_No := 402;
   Para[128].D_Address := 15152;
   Para[129].S_Line := 1;
   Para[129].S_ASDU := 29188;
   Para[129].S_Info := 6;
   Para[129].D_DB_No := 402;
   Para[129].D_Address := 15232;
   Para[130].S_Line := 1;
   Para[130].S_ASDU := 29188;
   Para[130].S_Info := 7;
   Para[130].D_DB_No := 402;
   Para[130].D_Address := 15312;
   Para[131].S_Line := 1;
   Para[131].S_ASDU := 30468;
   Para[131].S_Info := 240;
   Para[131].D_DB_No := 402;
   Para[131].D_Address := 15808;
   Para[132].S_Line := 1;
   Para[132].S_ASDU := 30468;
   Para[132].S_Info := 241;
   Para[132].D_DB_No := 402;
   Para[132].D_Address := 15888;
   Para[133].S_Line := 1;
   Para[133].S_ASDU := 30468;
   Para[133].S_Info := 242;
   Para[133].D_DB_No := 402;
   Para[133].D_Address := 15968;
   Para[134].S_Line := 1;
   Para[134].S_ASDU := 30468;
   Para[134].S_Info := 243;
   Para[134].D_DB_No := 402;
   Para[134].D_Address := 16048;
   Para[135].S_Line := 1;
   Para[135].S_ASDU := 30468;
   Para[135].S_Info := 2;
   Para[135].D_DB_No := 402;
   Para[135].D_Address := 16128;
   Para[136].S_Line := 1;
   Para[136].S_ASDU := 30468;
   Para[136].S_Info := 3;
   Para[136].D_DB_No := 402;
   Para[136].D_Address := 16208;
   Para[137].S_Line := 1;
   Para[137].S_ASDU := 30468;
   Para[137].S_Info := 4;
   Para[137].D_DB_No := 402;
   Para[137].D_Address := 16288;
   Para[138].S_Line := 1;
   Para[138].S_ASDU := 30468;
   Para[138].S_Info := 5;
   Para[138].D_DB_No := 402;
   Para[138].D_Address := 16368;
   Para[139].S_Line := 1;
   Para[139].S_ASDU := 30468;
   Para[139].S_Info := 6;
   Para[139].D_DB_No := 402;
   Para[139].D_Address := 16448;
   Para[140].S_Line := 1;
   Para[140].S_ASDU := 30468;
   Para[140].S_Info := 7;
   Para[140].D_DB_No := 402;
   Para[140].D_Address := 16528;
   Para[141].S_Line := 1;
   Para[141].S_ASDU := 5126;
   Para[141].S_Info := 240;
   Para[141].D_DB_No := 402;
   Para[141].D_Address := 17024;
   Para[142].S_Line := 1;
   Para[142].S_ASDU := 5126;
   Para[142].S_Info := 241;
   Para[142].D_DB_No := 402;
   Para[142].D_Address := 17104;
   Para[143].S_Line := 1;
   Para[143].S_ASDU := 5126;
   Para[143].S_Info := 242;
   Para[143].D_DB_No := 402;
   Para[143].D_Address := 17184;
   Para[144].S_Line := 1;
   Para[144].S_ASDU := 5126;
   Para[144].S_Info := 243;
   Para[144].D_DB_No := 402;
   Para[144].D_Address := 17264;
   Para[145].S_Line := 1;
   Para[145].S_ASDU := 5126;
   Para[145].S_Info := 2;
   Para[145].D_DB_No := 402;
   Para[145].D_Address := 17344;
   Para[146].S_Line := 1;
   Para[146].S_ASDU := 5126;
   Para[146].S_Info := 3;
   Para[146].D_DB_No := 402;
   Para[146].D_Address := 17424;
   Para[147].S_Line := 1;
   Para[147].S_ASDU := 5126;
   Para[147].S_Info := 4;
   Para[147].D_DB_No := 402;
   Para[147].D_Address := 17504;
   Para[148].S_Line := 1;
   Para[148].S_ASDU := 5126;
   Para[148].S_Info := 5;
   Para[148].D_DB_No := 402;
   Para[148].D_Address := 17584;
   Para[149].S_Line := 1;
   Para[149].S_ASDU := 5126;
   Para[149].S_Info := 6;
   Para[149].D_DB_No := 402;
   Para[149].D_Address := 17664;
   Para[150].S_Line := 1;
   Para[150].S_ASDU := 5126;
   Para[150].S_Info := 7;
   Para[150].D_DB_No := 402;
   Para[150].D_Address := 17744;

END_DATA_BLOCK

DATA_BLOCK "DB_IEC_Para_MAi_SC"
{ S7_Optimized_Access := 'FALSE' }
AUTHOR : SIE_GST
FAMILY : S7_IEC
NAME : P_CMD
VERSION : 1.6
   STRUCT
      DB_Manag { ExternalVisible := 'False'} : Struct
         Pos_of_DB { ExternalVisible := 'False'} : Byte;   // reserved for future - do not change !
         No_of_all_DBs { ExternalVisible := 'False'} : Byte;   // reserved for future - do not change !
         DB_No_Act { ExternalVisible := 'False'} : Word;   // reserved for future - do not change !
         DB_No_Prev { ExternalVisible := 'False'} : Word;   // reserved for future - do not change !
         DB_No_Next { ExternalVisible := 'False'} : Word;   // reserved for future - do not change !
         Reserved { ExternalVisible := 'False'} : Word;
      END_STRUCT;
      Info_Manag { ExternalVisible := 'False'} : Struct
         P_Byte_First_Info { ExternalVisible := 'False'} : Int;   // (Byte-) Position of first Para-Block - do not change !
         No_of_Infos { ExternalVisible := 'False'} : Int;   // 0:unspecified (DB is filled up to the end); otherwise size n of ARRAY [1..n]
         Len_Info { ExternalVisible := 'False'} : USInt;   // Difference in [byte] between two Para-Blocks - do not change !
         Len_Sort_Key { ExternalVisible := 'False'} : USInt;   // 0: without sorting; 1-8: Data sets are sorted ascending
         Re_internal_usage { ExternalVisible := 'False'} : DWord;
      END_STRUCT;
      Para_CMD { ExternalVisible := 'False'} : Array[1..30] of Struct
         S_DB_No { ExternalVisible := 'False'} : Int;   // Source:  No. of DB
         S_Adress { ExternalVisible := 'False'} : DInt;   // Source:  Bitposition
         D_Line { ExternalVisible := 'False'} : USInt;   // Dest. : No of Line (Nr der Linie) (1..x)-actually do not change from 1
         D_ASDU { ExternalVisible := 'False'} : UInt;   // Dest. : Address of ASDU (ASDU-Adresse)
         D_Info { ExternalVisible := 'False'} : DInt;   // Dest. : Address of Infoobject (IOA)
         Timeout { ExternalVisible := 'False'} : USInt;   // Timeout [sec] beginning with entry into send buffer...
         TI { ExternalVisible := 'False'} : USInt;   // Type Identifier 45(2Dhex=SC); 46(2E=DC); 47(2F=RC); 58,59,60 ->with time stamp
         Value { ExternalVisible := 'False'} : DWord;   // SCO/DCO/RCO-Byte, including Value-Bits (SCS/DCS/RCS),Qualifier (QU) and S/E-Bit
         Termination_Type { ExternalVisible := 'False'} : USInt;   // how a command will terminated (0:with sending;1:with recv.conf,2:with recv.term
         CMD_Info_Count { ExternalVisible := 'False'} : USInt;   // Only for reading: will incremented with each started command
         CMD_Info_State { ExternalVisible := 'False'} : Word;   // Only for reading: shows details of the last command process
      END_STRUCT;
   END_STRUCT;


